// TwinCAT 3 PLC project TwinCAT_OpenFramework_Tests
// Title: TwinCAT Open Framework Tests
// Company: Oleksandr Tiutyk FOP
// Author: Oleksandr Tiutyk
// ProjectVersion: 1.0.13.0
// Description: TwinCAT.OpenFramework regression tests and independent testing framework contract checks
// ProgramVersion: 3.1.4026.28
// libraries:
//   Tc2_Utilities, * (Beckhoff Automation GmbH)
//   [TwinCAT Open Framework JSON], * (Oleksandr Tiutyk FOP)
//   Tc3_JsonXml, * (Beckhoff Automation GmbH)
//   [TwinCAT Open Framework Testing], * (Oleksandr Tiutyk FOP)
//   Tc2_Standard, * (Beckhoff Automation GmbH)
//   Tc2_System, * (Beckhoff Automation GmbH)
//   [TwinCAT Open Framework Devices IO], * (Oleksandr Tiutyk FOP)
//   [TwinCAT Open Framework IO Models], * (Oleksandr Tiutyk FOP)
//   [TwinCAT Open Framework Automation], * (Oleksandr Tiutyk FOP)
//   [TwinCAT Open Framework Collections], * (Oleksandr Tiutyk FOP)
//   [TwinCAT Open Framework Comparison], * (Oleksandr Tiutyk FOP)
//   [TwinCAT Open Framework Core], * (Oleksandr Tiutyk FOP)
//   [TwinCAT Open Framework File System], * (Oleksandr Tiutyk FOP)
//   [TwinCAT Open Framework Loggers], * (Oleksandr Tiutyk FOP)
//   [TwinCAT Open Framework Timers], * (Oleksandr Tiutyk FOP)
//   [TwinCAT Open Framework Tasks], * (Oleksandr Tiutyk FOP)
//   [TwinCAT Open Framework Workflow], * (Oleksandr Tiutyk FOP)
// project tree:
//   Tests/Workflow/ WorkflowBindingTask.TcPOU, ComprehensiveTestWorkflow.TcPOU, RecoveryCatchTestActivity.TcPOU, ThrowingTestActivity.TcPOU, WORKFLOW_COMPREHENSIVE_TEST_SCENARIO.TcDUT, WorkflowComprehensiveTestGroup.TcPOU, WorkflowComprehensiveTestCase.TcPOU, WorkflowComprehensiveTestFixture.TcPOU, WorkflowContractActivity.TcPOU, WorkflowContractWorkflow.TcPOU, WorkflowContractTask.TcPOU, DELAY_PAUSE_TEST_PHASE.TcDUT, WORKFLOW_CONTRACT_TEST_SCENARIO.TcDUT, WorkflowContractTestGroup.TcPOU, WorkflowContractTestCase.TcPOU, WorkflowDelayPauseRemainingTest.TcPOU, WorkflowContractTestFixture.TcPOU
//   / CurrentNamespace.TcGVL, LogFilter.TcPOU, TestAutomationController.TcPOU, MAIN.TcPOU, TestTask.TcTTO, RunnerTestTask.TcTTO
//   Tests/JSON/ JSON_TEST_VALUE.TcDUT, JSON_TEST_SINGLE_VALUE.TcDUT, JSON_TEST_LARGE_VALUE.TcDUT, JsonExtenderProbe.TcPOU, AutomaticJsonRoundTripsAnyStructureTest.TcPOU, AutomaticJsonThrowingAnyRoundTripTest.TcPOU, AutomaticJsonSingleFieldVarInfoRoundTripTest.TcPOU, AutomaticJsonRejectsInvalidArgumentsTest.TcPOU, AutomaticJsonThrowingArgumentCategoriesTest.TcPOU, AutomaticJsonMalformedJsonAndReuseTest.TcPOU, AutomaticJsonWrappedCallbacksTest.TcPOU, AutomaticJsonCallbackContainmentAndReuseTest.TcPOU, AutomaticJsonThrowingCallbackPropagationTest.TcPOU, AutomaticJsonCapacityOverflowAndReuseTest.TcPOU, AutomaticJsonLongUtf8RoundTripTest.TcPOU, AutomaticJsonDecimalPlacesReadbackTest.TcPOU, AutomaticJsonSerializerTestGroup.TcPOU, MockConfigurationWritable.TcPOU, JsonConfigurationWriterTest.TcPOU, JsonConfigurationReaderTest.TcPOU, JsonConfigurationRoundTripTest.TcPOU, JsonConfigurationTestRunner.TcPOU
//   Tests/Collections/Contract/ CollectionCloneProbe.TcPOU, CollectionValidatorProbe.TcPOU, CollectionEqualityProbe.TcPOU, CollectionPredicateProbe.TcPOU, CollectionComparerProbe.TcPOU, COLLECTIONS_CONTRACT_SCENARIO.TcDUT, CollectionsContractTestFixture.TcPOU, CollectionsContractTestCase.TcPOU, CollectionsContractTestGroup.TcPOU, ICollectionSortValue.TcIO, CollectionComparableProbe.TcPOU
//   Tests/Collections/ DictionarySetAndGetTest.TcPOU, DictionaryRemoveTest.TcPOU, DictionaryContainsTest.TcPOU, ByteListTestCase.TcPOU, ByteListLoadFromAnyTest.TcPOU, ByteListIndexedAccessTest.TcPOU, ByteListFindTest.TcPOU, ByteListRemoveValueTest.TcPOU, ByteListRemoveRangeTest.TcPOU, ByteListClearTest.TcPOU, ListAppendTest.TcPOU, ListInsertTest.TcPOU, ListGetAndSetTest.TcPOU, ListFindTest.TcPOU, ListContainsTest.TcPOU, ListContainsGenericTest.TcPOU, ListRemoveFirstTest.TcPOU, ListRemoveMatchedTest.TcPOU, ListRemoveAtTest.TcPOU, ListSwapTest.TcPOU, ListAppendGenericTest.TcPOU, ListInsertGenericTest.TcPOU, ListGetAndSetGenericTest.TcPOU, ListStringPredicate.TcPOU, UniqueDataSetSetAndGetTest.TcPOU, UniqueDataSetRemoveTest.TcPOU, UniqueDataSetContainsTest.TcPOU, StackOwnedObjectCleanupTest.TcPOU, StackValidatorRejectionTest.TcPOU, StackIndexedAccessAndEnumerationTest.TcPOU, StackEmptyAndIndexBoundsTest.TcPOU, StackCopiedAndBorrowedValuesTest.TcPOU, StackContainsTest.TcPOU, StackContainsGenericTest.TcPOU, StackPushAndPeekTest.TcPOU, StackRemoveLastTest.TcPOU
//   Tests/Collections/Dynamic/ DynamicDictionaryClearTest.TcPOU, DynamicDictionaryTestGroup.TcPOU, DynamicByteListTestGroup.TcPOU, DynamicListSortTest.TcPOU, DynamicListClearTest.TcPOU, DynamicListTestGroup.TcPOU, DynamicUniqueDataSetClearTest.TcPOU, DynamicUniqueDataSetTestGroup.TcPOU, DynamicQueueContainsTest.TcPOU, DynamicQueueContainsGenericTest.TcPOU, DynamicQueueEnqueueAndPeekTest.TcPOU, DynamicQueueClearTest.TcPOU, DynamicQueueRemoveFirstTest.TcPOU, DynamicQueueTestGroup.TcPOU, DynamicStackClearTest.TcPOU, DynamicStackGrowthAndInvalidIncrementTest.TcPOU, DynamicStackTestGroup.TcPOU
//   Tests/Collections/Static/ StaticByteListOverflowTest.TcPOU, StaticByteListTestGroup.TcPOU, StaticDictionaryClearTest.TcPOU, StaticDictionaryOverflowTest.TcPOU, StaticDictionaryTestGroup.TcPOU, StaticListSortTest.TcPOU, StaticListClearTest.TcPOU, StaticListOverflowTest.TcPOU, StaticListTestGroup.TcPOU, StaticUniqueDataSetClearTest.TcPOU, StaticUniqueDataSetOverflowTest.TcPOU, StaticUniqueDataSetTestGroup.TcPOU, StaticQueueContainsTest.TcPOU, StaticQueueContainsGenericTest.TcPOU, StaticQueueEnqueueAndPeekTest.TcPOU, StaticQueueClearTest.TcPOU, StaticQueueRemoveFirstTest.TcPOU, StaticQueueOverflowTest.TcPOU, StaticQueueTestGroup.TcPOU, StaticStackClearTest.TcPOU, StaticStackOverflowTest.TcPOU, StaticStackTestGroup.TcPOU
//   Tests/Devices/IO/ RangeAnalogValueConverterTest.TcPOU, RangeAnalogValueConverter16BitTest.TcPOU, RangeAnalogValueConverter32BitTest.TcPOU, RangeAnalogValueConverter32RealTest.TcPOU, AnalogInputConverterProbe.TcPOU, AnalogInputRecoveryProbe.TcPOU, DigitalInputNormallyOpenTest.TcPOU, DigitalInputNormallyClosedTest.TcPOU, DigitalInputUnboundTest.TcPOU, DigitalOutputNormallyOpenTest.TcPOU, DigitalOutputNormallyClosedTest.TcPOU, DirectAnalogValueConverterTest.TcPOU, AnalogInputScalingAndScalarBindingTest.TcPOU, AnalogInputChannelStatusAndErrorReportingTest.TcPOU, AnalogInputConverterRecoveryTest.TcPOU, AnalogInputCriticalConversionErrorTest.TcPOU, AnalogInputStatusWordIsolationTest.TcPOU, AnalogInputStatusBitDecodingTest.TcPOU, AnalogOutputScalingTest.TcPOU, AnalogOutputEqualRawLimitsTest.TcPOU, DynamicRangeAnalogValueConverterTest.TcPOU, StaticConverterCopiesLimitsTest.TcPOU, RangeConverterBoundaryClampingAndZeroDivisionTest.TcPOU, DevicesIOTestGroup.TcPOU, IO_MODELS_TEST_SCENARIO.TcDUT, IIOModelsTestFixture.TcIO, IOModelsTestFixture.TcPOU, IOModelsTestCase.TcPOU, IOModelsTestGroup.TcPOU
//   Tests/Core/ NotImplementedExceptionTest.TcPOU, StandardExceptionChainTest.TcPOU, AggregateExceptionPropagationTest.TcPOU, SavedFrameworkExceptionRethrowTest.TcPOU, SystemExceptionRethrowTest.TcPOU, ExceptionTimestampFormattingTest.TcPOU, SystemExceptionTimestampFormattingTest.TcPOU, SystemExceptionCloneTest.TcPOU, AggregateExceptionCloneTest.TcPOU, ArgumentTypeExceptionCloneTest.TcPOU, ExceptionGraphRejectionTest.TcPOU, AggregateExceptionBoundedMessageTest.TcPOU, ExceptionTestGroup.TcPOU, ObjectExitProbe.TcPOU, GenericLongStringOrderingTest.TcPOU, GenericStringPrefixOrderingTest.TcPOU, GenericNaNOrderingTest.TcPOU, GenericMixedNumericPrecisionTest.TcPOU, GenericConversionPairsTest.TcPOU, SystemTypeClassFormattingTest.TcPOU, SystemTypeClassDiagnosticsTest.TcPOU, GenericBorrowedWritesTest.TcPOU, GenericValueTestGroup.TcPOU, DynamicObjectDisposalTest.TcPOU, ObjectInterfaceAddressTest.TcPOU, StaticObjectReleaseRefusalTest.TcPOU, ObjectLifetimeTestGroup.TcPOU, ExceptionTimestampProbe.TcPOU, RandomRangeTest.TcPOU, RandomAbsoluteDispersionTest.TcPOU, RandomPercentageDispersionTest.TcPOU, RandomTestGroup.TcPOU
//   Tests/Files/ FileManagerStartRefusalProbe.TcPOU, FILE_CALLER_CLEANUP_TEST_PHASE.TcDUT, FILE_OPERATIONS_TEST_PHASE.TcDUT, FILE_BUFFER_TEST_PHASE.TcDUT, FileSystemIntegrationTestGroup.TcPOU, FileByteOperationsTest.TcPOU, FileBinaryBufferMatrixTest.TcPOU, FileCallerExceptionCleanupTest.TcPOU, FileSystemContractTest.TcPOU, FileSystemDefaultNamesTest.TcPOU, FileSystemUnboundContentTest.TcPOU, FileSystemLoadBufferTest.TcPOU, FileSystemQueueBindingTest.TcPOU, FileSystemExceptionCloneTest.TcPOU, FileSystemManagerStartRefusalTest.TcPOU, LexicalPathValidationTest.TcPOU, PATH_VALIDATION_TEST_CASE.TcDUT, FileTestRoot.TcPOU, FILE_TEST_DIRECTORY_PHASE.TcDUT, FileTestDirectory.TcPOU, DIRECTORY_TEST_STEP.TcDUT, DirectoryTest.TcPOU, DirectoryOperationTest.TcPOU, READ_ONLY_FILE_TEST_STEP.TcDUT, FILE_MANAGER_REUSE_TEST_STEP.TcDUT, FILE_TEST_LIFECYCLE.TcDUT, FileContentScenarioTest.TcPOU, FileTextReadWriteTest.TcPOU, FileReadOnlyWriteTest.TcPOU, FileWriteCancellationTest.TcPOU, FileManagerReuseTest.TcPOU, FileContentManagerOperationsTest.TcPOU, OpenMissingFileForReadingTest.TcPOU
//   Tests/Loggers/ LOGGER_DELIVERY_BEHAVIOR.TcDUT, LOGGER_CAPTURED_MESSAGE.TcDUT, LoggerCaptureBackend.TcPOU, LoggerTaskProbe.TcPOU, QueuedLoggerSnapshotTest.TcPOU, LoggerIntegrationTestGroup.TcPOU, EventLoggerCategoryTest.TcPOU, QueuedEventLoggerTest.TcPOU, TextFileLoggerRotationTest.TcPOU, QueuedLoggerCapacityTest.TcPOU, QueuedLoggerDeliveryFailureTest.TcPOU, LoggerFormatterFailureTest.TcPOU, LoggerMetadataAndRecordLimitTest.TcPOU, LoggerTaskDiagnosticsTest.TcPOU, QueuedLoggerAggregateTest.TcPOU, CurrentTaskLoggerRoutingTest.TcPOU, LoggerNonCyclicInitializationTest.TcPOU, LoggerContractTestGroup.TcPOU, LOGGER_DIRECTORY_CLEANUP_PHASE.TcDUT, LoggerTestDirectory.TcPOU, LOGGER_FILE_TEST_PHASE.TcDUT, LoggerRoutingTest.TcPOU
//   Tests/Strings/String/ StringBuilderEmptyTest.TcPOU, StringBuilderContentTest.TcPOU, StringBuilderAssignmentFailureTest.TcPOU, StringBuilderTestGroup.TcPOU, StringFitFormattingTest.TcPOU, StringAppendTest.TcPOU, StringAppendFitTest.TcPOU, StringConcatFitTest.TcPOU, StringContainsTest.TcPOU, StringJoinTest.TcPOU, StringReplacementTest.TcPOU, StringSplitTest.TcPOU, StringTrimTest.TcPOU, StringSeparatorBoundsTest.TcPOU, StringsTestGroup.TcPOU
//   Tests/Strings/WideString/ WideStringBuilderEmptyTest.TcPOU, WideStringBuilderContentTest.TcPOU, WideStringBuilderAssignmentFailureTest.TcPOU, WideStringBuilderTestGroup.TcPOU, WideStringFitFormattingTest.TcPOU, WideStringAppendTest.TcPOU, WideStringAppendFitTest.TcPOU, WideStringConcatFitTest.TcPOU, WideStringContainsTest.TcPOU, WideStringJoinTest.TcPOU, WideStringReplacementTest.TcPOU, WideStringSplitTest.TcPOU, WideStringTrimTest.TcPOU, WideStringSeparatorBoundsTest.TcPOU, WideStringLongFitFormattingTest.TcPOU, WideStringsTestGroup.TcPOU
//   Tests/Tasks/QueueCleanup/ QueueCleanupChild.TcPOU, QueueCleanupQueue.TcPOU, QueueCleanupResource.TcPOU, ThrowingGetMessageException.TcPOU, QUEUE_CLEANUP_TEST_SCENARIO.TcDUT, QUEUE_CLEANUP_TEST_PHASE.TcDUT, TaskQueueCleanupScenarioTest.TcPOU, TaskQueueCleanupTestGroup.TcPOU
//   Tests/Tasks/Sequence/ CounterTask.TcPOU, TaskSequenceFifoTest.TcPOU, TaskQueueEmptyModeTest.TcPOU, TaskSequenceTestGroup.TcPOU
//   Tests/Tasks/Stopping/ TaskStoppingResource.TcPOU, TaskStoppingProbe.TcPOU, TASK_STOPPING_TEST_SCENARIO.TcDUT, TaskStoppingScenarioTest.TcPOU, TaskStoppingTestGroup.TcPOU, TaskStoppingNameTest.TcPOU, TimerRestartProbe.TcPOU, PrepareTimerTestForReuse.TcPOU, TimerMetadataTest.TcPOU, TimerCancelBeforeExecuteTest.TcPOU, TimerResetAfterCompletionTest.TcPOU, TimerPendingRestartTest.TcPOU, TimerRestartResetFailureTest.TcPOU, TimerRestartStartFailureTest.TcPOU, TimerCompletionCallbackTest.TcPOU, TimerCompletionPulseTest.TcPOU, DELAYED_TIMER_TEST_SCENARIO.TcDUT, DelayedTimerObservationTest.TcPOU, TimerIntervalObservationTest.TcPOU, TimerTimingTestGroup.TcPOU, TimerRestartWhileRunningTest.TcPOU
//   Tests/Testing/ AssertionCallerTestRunner.TcPOU, AssertionTestRunner.TcPOU, DeadlineTestRunner.TcPOU, DiagnosticTestRunner.TcPOU, EmptyTestRunner.TcPOU, ExternalRecoveryTestRunner.TcPOU, IsolationTestRunner.TcPOU, MissingChildrenTestRunner.TcPOU, MixedTestRunner.TcPOU, ReporterAbortTestRunner.TcPOU, RootTopologyTestRunner.TcPOU, AssertionIsolationProbe.TcPOU, TestingProbe.TcPOU, ThrowingTestReporter.TcPOU, CapturingAdsLogReporter.TcPOU, ExternalElementProbe.TcPOU, DiagnosticProbe.TcPOU, ASSERTION_PROBE_SCENARIO.TcDUT, AssertionContractProbe.TcPOU, EmptyTestGroup.TcPOU, SingleChildTestGroup.TcPOU, PairTestGroup.TcPOU, FailureTestGroup.TcPOU, NestedFailureTestGroup.TcPOU, DeadlineTestGroup.TcPOU, MissingChildrenTestGroup.TcPOU, TEST_RUNNER_CONTRACT_SCENARIO.TcDUT, TestRunnerContractTest.TcPOU
//   Tests/Tasks/ UnboundTaskStateTest.TcPOU, BoundTaskStateTest.TcPOU, UnboundTaskRunningSubstateTest.TcPOU, BoundTaskRunningSubstateTest.TcPOU, UnboundTaskStopReasonTest.TcPOU, BoundTaskStopReasonTest.TcPOU, TaskReinitViewsTest.TcPOU, TaskNamePreservedByResetTest.TcPOU, TaskLifecycleViewsTestGroup.TcPOU
//   Tests/Automation/ AUTOMATION_COMPONENT_TEST_SCENARIO.TcDUT, AutomationComponentTestGroup.TcPOU, AutomationComponentTestCase.TcPOU, AutomationChildInitializationTimeoutTest.TcPOU, AutomationRunnerObservationTest.TcPOU, AutomationComponentTestFixture.TcPOU, RUNNER_TEST_PHASE.TcDUT, AutomationRunnerTestProgram.TcPOU, AutomationRunnerTestGlobals.TcGVL, MockPluginAutomationController.TcPOU, MockHmiControllerPlugin.TcPOU, MockAutomationController.TcPOU, MockAutomationEvent.TcPOU, MockCompositeAutomationComponent.TcPOU, MockLeafAutomationComponent.TcPOU
//   Version/ Global_Version.TcGVL
// (motion and I/O tree: see PLC project twincat_openframework_core)
// real-time tasks:
//   TASK PlcTask: cycle T#10ms, priority 20, ADS port 350
//   TASK TestTask: cycle T#10ms, priority 1, ADS port 351
//   TASK RunnerTestTask: cycle T#10ms, priority 2, ADS port 354
//   TASK HowToTask: cycle T#10ms, priority 22, ADS port 353
// variable links:

CONFIGURATION TwinCAT_OpenFramework_Tests
    RESOURCE PLC ON TwinCAT3
        TASK TestTask(INTERVAL := T#10ms, PRIORITY := 1);
        TASK RunnerTestTask(INTERVAL := T#10ms, PRIORITY := 2);
        PROGRAM MAIN WITH TestTask : MAIN;
        PROGRAM AutomationRunnerTestProgram WITH RunnerTestTask : AutomationRunnerTestProgram;
    END_RESOURCE
END_CONFIGURATION

// ---- Tests/JSON/JSON_TEST_VALUE.TcDUT
(*
SPDX-FileCopyrightText: © 2026 Oleksandr Tiutyk <trofimich@gmail.com>
SPDX-License-Identifier: MIT
License: https://opensource.org/license/mit
*)

(*!
<summary>Holds a multi-field live value for native JSON round-trip tests.</summary>
*)
TYPE JSON_TEST_VALUE :
STRUCT
	//! <summary>Integer payload with an independent expected value.</summary>
	Number : DINT;
	//! <summary>Boolean payload used to detect incomplete restoration.</summary>
	Ready : BOOL;
END_STRUCT
END_TYPE

// ---- Tests/JSON/JSON_TEST_SINGLE_VALUE.TcDUT
(*
SPDX-FileCopyrightText: © 2026 Oleksandr Tiutyk <trofimich@gmail.com>
SPDX-License-Identifier: MIT
License: https://opensource.org/license/mit
*)

(*!
<summary>Holds a single-field structure for explicit VAR_INFO type resolution.</summary>
*)
TYPE JSON_TEST_SINGLE_VALUE :
STRUCT
	//! <summary>Value restored through the explicit structure type.</summary>
	Number : DINT;
END_STRUCT
END_TYPE

// ---- Tests/JSON/JSON_TEST_LARGE_VALUE.TcDUT
(*
SPDX-FileCopyrightText: © 2026 Oleksandr Tiutyk <trofimich@gmail.com>
SPDX-License-Identifier: MIT
License: https://opensource.org/license/mit
*)

(*!
<summary>Holds long text and a distinct marker for native capacity and encoding tests.</summary>
*)
TYPE JSON_TEST_LARGE_VALUE :
STRUCT
	//! <summary>Uses the framework JSON text capacity in bytes, excluding the terminator.</summary>
	Text : STRING(TOF_Core.Parameters.JSON_DOCUMENT_CHAR_SIZE);
	//! <summary>Independent field that distinguishes the structure from its first member.</summary>
	Marker : DINT;
END_STRUCT
END_TYPE

// ---- Tests/Collections/Contract/COLLECTIONS_CONTRACT_SCENARIO.TcDUT
(*!
<summary>Selects one scenario in the collection contract group.</summary>
<description>
Each value maps to a separately reported single-cycle case.
</description>
*)
{attribute 'qualified_only'}
{attribute 'strict'}
TYPE COLLECTIONS_CONTRACT_SCENARIO :
(
	COPY_FAILURE_PRESERVES_EXCEPTION,
	SECOND_COPY_FAILURE_CLEANUP,
	STATIC_FULL_COPY_CLEANUP,
	BYTE_OVERLAP_AND_BOUNDS,
	BYTE_SIZE_REJECTIONS,
	LIST_OWNERSHIP_REPLACEMENT,
	LIST_REMOVAL_LIMITS,
	SORT_FAILURE_PRESERVES_ENTRIES,
	QUEUE_VALIDATION_AND_GROWTH,
	HASH_COLLISION_GROWTH,
	HASH_EQUALITY_REPRESENTATIONS,
	HASH_OWNERSHIP_ALIASES,
	FULL_STATIC_DUPLICATE_UPDATES,
	QUERY_FAILURE_CLEANUP,
	CONTAINS_COLLECTION_CALLBACK_FAILURES,
	GENERIC_QUERY_RELEASE_MATRIX,
	ALL_CURSOR_CONTRACTS,
	FIXTURE_CLEANUP_AFTER_EXCEPTION,
	DEFAULT_SORT_NUMERIC_BRANCHES,
	DEFAULT_SORT_TEXT_AND_OBJECTS,
	DEFAULT_SORT_EXPLICIT_AND_REJECTION,
	MISSING_CURSOR_SOURCES
);
END_TYPE

// ---- Tests/Devices/IO/IO_MODELS_TEST_SCENARIO.TcDUT
(*!
<summary>Selects one independently reported IO model test scenario.</summary>
*)
{attribute 'qualified_only'}
{attribute 'strict'}
TYPE IO_MODELS_TEST_SCENARIO :
(
	PULSE_TRAIN,
	ENCODER_CHANNELS,
	POWER_MEASUREMENT,
	AUXILIARY,
	COUNTER_AND_LOAD,
	SERIAL_AND_DIAGNOSTICS,
	DISCRETE_CATALOG,
	ANALOG_REPRESENTATIONS,
	DINT_BINDING,
	REAL_BINDING
);
END_TYPE

// ---- Tests/Files/FILE_CALLER_CLEANUP_TEST_PHASE.TcDUT
(*
SPDX-FileCopyrightText: © 2026 Oleksandr Tiutyk <trofimich@gmail.com>
SPDX-License-Identifier: MIT
License: https://opensource.org/license/mit
*)

(*!
<summary>Names the phases of a caught caller-exception cleanup regression.</summary>
*)
{attribute 'qualified_only'}
{attribute 'strict'}
TYPE FILE_CALLER_CLEANUP_TEST_PHASE :
(
	//! <summary>Prepare an exclusively owned scenario directory.</summary>
	PREPARE_DIRECTORY,
	//! <summary>Open a file and leave the manager waiting for future children.</summary>
	OPEN_FILE,
	//! <summary>Observe acquisition and raise a caller-side exception.</summary>
	INJECT_CALLER_EXCEPTION,
	//! <summary>Continue cancellation and stopping after the exception was caught.</summary>
	DRAIN_MANAGER,
	//! <summary>Remove owned artifacts only after release completed.</summary>
	CLEANUP
);
END_TYPE

// ---- Tests/Files/FILE_OPERATIONS_TEST_PHASE.TcDUT
(*
SPDX-FileCopyrightText: © 2026 Oleksandr Tiutyk <trofimich@gmail.com>
SPDX-License-Identifier: MIT
License: https://opensource.org/license/mit
*)

(*!
<summary>Names the phases of a filesystem integration regression.</summary>
*)
{attribute 'qualified_only'}
{attribute 'strict'}
TYPE FILE_OPERATIONS_TEST_PHASE :
(
	//! <summary>prepare directory.</summary>
	PREPARE_DIRECTORY,
	//! <summary>start write.</summary>
	START_WRITE,
	//! <summary>wait for write.</summary>
	WAIT_FOR_WRITE,
	//! <summary>check collisions.</summary>
	CHECK_COLLISIONS,
	//! <summary>wait for collisions.</summary>
	WAIT_FOR_COLLISIONS,
	//! <summary>start load.</summary>
	START_LOAD,
	//! <summary>wait for load.</summary>
	WAIT_FOR_LOAD,
	//! <summary>start rename.</summary>
	START_RENAME,
	//! <summary>wait for rename.</summary>
	WAIT_FOR_RENAME,
	//! <summary>load renamed file.</summary>
	LOAD_RENAMED_FILE,
	//! <summary>wait for renamed load.</summary>
	WAIT_FOR_RENAMED_LOAD,
	//! <summary>start delete.</summary>
	START_DELETE,
	//! <summary>wait for delete.</summary>
	WAIT_FOR_DELETE,
	//! <summary>load deleted file.</summary>
	LOAD_DELETED_FILE,
	//! <summary>wait for missing load.</summary>
	WAIT_FOR_MISSING_LOAD,
	//! <summary>cleanup.</summary>
	CLEANUP
);
END_TYPE

// ---- Tests/Files/FILE_BUFFER_TEST_PHASE.TcDUT
(*
SPDX-FileCopyrightText: © 2026 Oleksandr Tiutyk <trofimich@gmail.com>
SPDX-License-Identifier: MIT
License: https://opensource.org/license/mit
*)

(*!
<summary>Names the phases of a filesystem integration regression.</summary>
*)
{attribute 'qualified_only'}
{attribute 'strict'}
TYPE FILE_BUFFER_TEST_PHASE :
(
	//! <summary>prepare directory.</summary>
	PREPARE_DIRECTORY,
	//! <summary>create file.</summary>
	CREATE_FILE,
	//! <summary>wait for file.</summary>
	WAIT_FOR_FILE,
	//! <summary>start invalid operation.</summary>
	START_INVALID_OPERATION,
	//! <summary>wait for invalid operation.</summary>
	WAIT_FOR_INVALID_OPERATION,
	//! <summary>cleanup.</summary>
	CLEANUP
);
END_TYPE

// ---- Tests/Files/PATH_VALIDATION_TEST_CASE.TcDUT
(*
SPDX-FileCopyrightText: © 2026 Oleksandr Tiutyk <trofimich@gmail.com>
SPDX-License-Identifier: MIT
License: https://opensource.org/license/mit
*)

(*!
<summary>Pairs a path with its expected lexical outcomes for directory and file validation.</summary>
*)
TYPE PATH_VALIDATION_TEST_CASE :
STRUCT
	//! <summary>Null-terminated path passed to each lexical validator.</summary>
	Path : Tc2_System.T_MaxString;
	//! <summary>Expected result from IsValidDirectoryPath.</summary>
	DirectoryAccepted : BOOL;
	//! <summary>Expected result from IsValidFilePath.</summary>
	FileAccepted : BOOL;
END_STRUCT
END_TYPE

// ---- Tests/Files/FILE_TEST_DIRECTORY_PHASE.TcDUT
(*
SPDX-FileCopyrightText: © 2026 Oleksandr Tiutyk <trofimich@gmail.com>
SPDX-License-Identifier: MIT
License: https://opensource.org/license/mit
*)

(*!
<summary>Names preparation and cleanup phases of one exclusively owned file-test directory.</summary>
*)
{attribute 'qualified_only'}
{attribute 'strict'}
TYPE FILE_TEST_DIRECTORY_PHASE :
(
	//! <summary>Create a new directory; an existing entry is a preparation failure.</summary>
	CREATE_DIRECTORY,
	//! <summary>Wait for ordinary creation before establishing ownership.</summary>
	WAIT_FOR_DIRECTORY,
	//! <summary>The scenario exclusively owns its prepared directory.</summary>
	READY,
	//! <summary>Cancel and drain interrupted preparation without guessing ownership.</summary>
	DRAIN_CREATION,
	//! <summary>Attempt deletion of the first registered scenario artifact.</summary>
	DELETE_FIRST_FILE,
	//! <summary>Attempt deletion of the second registered scenario artifact.</summary>
	DELETE_SECOND_FILE,
	//! <summary>Remove the owned directory nonrecursively after file cleanup attempts.</summary>
	REMOVE_DIRECTORY,
	//! <summary>Preparation failed or cleanup attempts finished; inspect result properties.</summary>
	COMPLETE
);
END_TYPE

// ---- Tests/Files/DIRECTORY_TEST_STEP.TcDUT
(*
SPDX-FileCopyrightText: © 2026 Oleksandr Tiutyk <trofimich@gmail.com>
SPDX-License-Identifier: MIT
License: https://opensource.org/license/mit
*)

(*!
<summary>Names the operations and successful completion of DirectoryTest scenarios.</summary>
<description>
Each scenario follows its explicit subset of steps. Advancing requires the expected stop reason and any
existence checks for that step. COMPLETED ends scenario work. Cleanup advances on later test cycles.
The enum is internal to the tests.
</description>
*)
{attribute 'qualified_only'}
{attribute 'strict'}
{attribute 'to_string'}
TYPE DIRECTORY_TEST_STEP :
(
	//! <summary>Create the test directory; success establishes ownership, an existing path causes failure.</summary>
	CREATE_DIRECTORY := 0,
	//! <summary>Verify the newly created test directory exists.</summary>
	CHECK_DIRECTORY_PRESENT,
	//! <summary>Create a child directory inside the owned test directory.</summary>
	CREATE_CHILD_DIRECTORY,
	//! <summary>Verify the first conditional creation produced a child directory.</summary>
	CHECK_CHILD_DIRECTORY_PRESENT,
	//! <summary>Repeat conditional creation while the child directory exists.</summary>
	CREATE_CHILD_DIRECTORY_AGAIN,
	//! <summary>Verify the child directory still exists after repeated creation.</summary>
	CHECK_CHILD_DIRECTORY_PRESENT_AGAIN,
	//! <summary>Require native removal of the nonempty parent directory to fail.</summary>
	REJECT_NONEMPTY_DIRECTORY_REMOVAL,
	//! <summary>Confirm the child still exists after the failed parent removal.</summary>
	CHECK_CHILD_DIRECTORY_RETAINED,
	//! <summary>Remove the owned child directory using conditional removal.</summary>
	REMOVE_CHILD_DIRECTORY,
	//! <summary>Verify that the child directory is absent.</summary>
	CHECK_CHILD_DIRECTORY_ABSENT,
	//! <summary>Repeat conditional removal while the child directory is absent.</summary>
	REMOVE_CHILD_DIRECTORY_AGAIN,
	//! <summary>Verify the child directory is still absent after repeated removal.</summary>
	CHECK_CHILD_DIRECTORY_ABSENT_AGAIN,
	//! <summary>Remove the empty test directory created by this scenario.</summary>
	REMOVE_DIRECTORY,
	//! <summary>Verify the test directory is absent after removal.</summary>
	CHECK_DIRECTORY_ABSENT,
	//! <summary>All scenario operations and postconditions completed successfully.</summary>
	COMPLETED
);
END_TYPE

// ---- Tests/Files/READ_ONLY_FILE_TEST_STEP.TcDUT
(*
SPDX-FileCopyrightText: © 2026 Oleksandr Tiutyk <trofimich@gmail.com>
SPDX-License-Identifier: MIT
License: https://opensource.org/license/mit
*)

(*!
<summary>Names preparation and write-failure checks for a file opened for reading.</summary>
<description>
Steps belong to one test scenario; values are not a serialized protocol. The first member is the initial
preparation step. Test completion and failure cleanup are tracked separately.
</description>
*)
{attribute 'qualified_only'}
{attribute 'strict'}
{attribute 'to_string'}
TYPE READ_ONLY_FILE_TEST_STEP :
(
	CREATE_FILE,
	OPEN_FILE_FOR_READING,
	CHECK_WRITE_FAILURE
);
END_TYPE

// ---- Tests/Files/FILE_MANAGER_REUSE_TEST_STEP.TcDUT
(*
SPDX-FileCopyrightText: © 2026 Oleksandr Tiutyk <trofimich@gmail.com>
SPDX-License-Identifier: MIT
License: https://opensource.org/license/mit
*)

(*!
<summary>Names the two runs and intervening cancellation in the file-manager reuse test.</summary>
<description>
Steps belong to one test scenario; values are not a serialized protocol. The first member is the initial
preparation step. Test completion and failure cleanup are tracked separately.
</description>
*)
{attribute 'qualified_only'}
{attribute 'strict'}
{attribute 'to_string'}
TYPE FILE_MANAGER_REUSE_TEST_STEP :
(
	START_FIRST_WRITE,
	CANCEL_AFTER_WRITE,
	RESET_AND_START_SECOND_FILE,
	CHECK_SECOND_FILE
);
END_TYPE

// ---- Tests/Files/FILE_TEST_LIFECYCLE.TcDUT
(*
SPDX-FileCopyrightText: © 2026 Oleksandr Tiutyk <trofimich@gmail.com>
SPDX-License-Identifier: MIT
License: https://opensource.org/license/mit
*)

(*!
<summary>Separates filesystem scenario execution from cleanup and result reporting.</summary>
<description>
A case remains active while cleanup is pending. Completed drain and cleanup attempts permit FINISHED
and result reporting. Errors remain test failures and do not authorize deleting unowned paths.
Cleanup has no forced deadline. These phases do not guarantee physical close after a native release failure.
</description>
*)
{attribute 'qualified_only'}
{attribute 'strict'}
TYPE FILE_TEST_LIFECYCLE :
(
	//! <summary>Advance the scenario and its deadline until its normal or failed outcome is known.</summary>
	RUNNING_SCENARIO,
	//! <summary>Keep the case active while retained resources stop and owned cleanup attempts finish.</summary>
	CLEANING_UP,
	//! <summary>Cleanup observations were reported for this run.</summary>
	FINISHED
);
END_TYPE

// ---- Tests/Loggers/LOGGER_DELIVERY_BEHAVIOR.TcDUT
(*
SPDX-FileCopyrightText: © 2026 Oleksandr Tiutyk <trofimich@gmail.com>
SPDX-License-Identifier: MIT
License: https://opensource.org/license/mit
*)
(*!
<summary>Selects the deliberate backend outcome used by logger containment tests.</summary>
*)
{attribute 'qualified_only'}
{attribute 'strict'}
TYPE LOGGER_DELIVERY_BEHAVIOR :
(
	ACCEPT,
	REFUSE,
	THROW_EXCEPTION
);
END_TYPE

// ---- Tests/Loggers/LOGGER_CAPTURED_MESSAGE.TcDUT
(*
SPDX-FileCopyrightText: © 2026 Oleksandr Tiutyk <trofimich@gmail.com>
SPDX-License-Identifier: MIT
License: https://opensource.org/license/mit
*)
(*!
<summary>Owns one captured logger call independently of caller buffers.</summary>
*)
TYPE LOGGER_CAPTURED_MESSAGE :
STRUCT
	Category : TOF_Core.LOG_CATEGORY;
	Message : TOF_Core.ERROR_MESSAGE;
	HasMessageNumber : BOOL;
	MessageNumber : ULINT;
END_STRUCT
END_TYPE

// ---- Tests/Loggers/LOGGER_DIRECTORY_CLEANUP_PHASE.TcDUT
(*
SPDX-FileCopyrightText: © 2026 Oleksandr Tiutyk <trofimich@gmail.com>
SPDX-License-Identifier: MIT
License: https://opensource.org/license/mit
*)
(*!
<summary>Identifies owned log discovery, byte readback, deletion and final directory cleanup.</summary>
*)
{attribute 'qualified_only'}
{attribute 'strict'}
TYPE LOGGER_DIRECTORY_CLEANUP_PHASE :
(
	ENUMERATE_FIRST,
	ENUMERATE_WAIT,
	ENUMERATE_NEXT,
	LOAD_FILE,
	WAIT_FOR_LOAD,
	DELETE_FILE,
	WAIT_FOR_DELETE,
	REMOVE_DIRECTORY,
	COMPLETE
);
END_TYPE

// ---- Tests/Loggers/LOGGER_FILE_TEST_PHASE.TcDUT
(*
SPDX-FileCopyrightText: © 2026 Oleksandr Tiutyk <trofimich@gmail.com>
SPDX-License-Identifier: MIT
License: https://opensource.org/license/mit
*)
(*!
<summary>Identifies owned directory preparation, logging, idle observation, stopping and readback phases.</summary>
*)
{attribute 'qualified_only'}
{attribute 'strict'}
TYPE LOGGER_FILE_TEST_PHASE :
(
	PREPARE_DIRECTORY,
	SEND_MESSAGES,
	OBSERVE_IDLE,
	WAIT_FOR_STOP,
	READBACK,
	COMPLETE
);
END_TYPE

// ---- Tests/Tasks/QueueCleanup/QUEUE_CLEANUP_TEST_SCENARIO.TcDUT
(*
SPDX-FileCopyrightText: © 2026 Oleksandr Tiutyk <trofimich@gmail.com>
SPDX-License-Identifier: MIT
License: https://opensource.org/license/mit
*)

(*!
<summary>Selects the faults and observations for a queue cleanup case.</summary>
*)
{attribute 'qualified_only'}
{attribute 'strict'}
TYPE QUEUE_CLEANUP_TEST_SCENARIO :
(
	//! <summary>Completes cleanup, then reuses the same queue and child without injection.</summary>
	DELAYED_CLEANUP_AND_REUSE,
	//! <summary>Raises two further exceptions on cleanup Execute calls.</summary>
	REPEATED_EXECUTE_FAILURE,
	//! <summary>Refuses cancellation by exception twice before accepting it.</summary>
	CANCEL_REQUEST_FAILURE,
	//! <summary>Raises a secondary exception while formatting the original failure.</summary>
	MESSAGE_FORMATTING_FAILURE,
	//! <summary>Requests owner cancellation after the first processing failure.</summary>
	EXTERNAL_CANCEL_DURING_CLEANUP,
	//! <summary>Holds cooperative child cleanup across eight subsequent queue calls.</summary>
	HELD_CLEANUP,
	//! <summary>Requests owner cancellation and injects a terminal parent release failure.</summary>
	EXTERNAL_CANCEL_WITH_RELEASE_FAILURE
);
END_TYPE

// ---- Tests/Tasks/QueueCleanup/QUEUE_CLEANUP_TEST_PHASE.TcDUT
(*
SPDX-FileCopyrightText: © 2026 Oleksandr Tiutyk <trofimich@gmail.com>
SPDX-License-Identifier: MIT
License: https://opensource.org/license/mit
*)

(*!
<summary>Identifies the current queue cleanup test phase.</summary>
*)
{attribute 'qualified_only'}
{attribute 'strict'}
TYPE QUEUE_CLEANUP_TEST_PHASE :
(
	//! <summary>Drive the original failure and child cleanup.</summary>
	FAILURE_RUN,
	//! <summary>Drive the same queue after Reset without a child failure.</summary>
	REUSE_RUN,
	//! <summary>Advance the stopped queue once to check that release is not retried.</summary>
	OBSERVE_FAILED_RELEASE
);
END_TYPE

// ---- Tests/Tasks/Stopping/TASK_STOPPING_TEST_SCENARIO.TcDUT
(*
SPDX-FileCopyrightText: © 2026 Oleksandr Tiutyk <trofimich@gmail.com>
SPDX-License-Identifier: MIT
License: https://opensource.org/license/mit
*)

(*!
<summary>Selects the injection and expected behavior of a task stopping case.</summary>
*)

{attribute 'qualified_only'}
{attribute 'strict'}
TYPE TASK_STOPPING_TEST_SCENARIO :
(
	//! <summary>Completes work and waits for both stopping and release.</summary>
	WORK_DONE,
	//! <summary>Retains the ERROR result and diagnostic after cleanup.</summary>
	WORK_ERROR,
	//! <summary>Retains the ABORTED result and diagnostic after cleanup.</summary>
	WORK_ABORT,
	//! <summary>Defers stopping after a processing exception.</summary>
	WORK_EXCEPTION,
	//! <summary>Uses a named fallback when the processing exception formatter throws.</summary>
	WORK_FORMATTER_EXCEPTION,
	//! <summary>Retries the interrupted stopping hook and preserves the preceding work exception.</summary>
	FIRST_STOPPING_EXCEPTION,
	//! <summary>Interrupts three stopping calls before allowing progress.</summary>
	REPEATED_STOPPING_EXCEPTIONS,
	//! <summary>Produces a named fallback for empty exception text without a bound resource.</summary>
	EMPTY_WORK_EXCEPTION_MESSAGE,
	//! <summary>Cancels a pending acquisition and releases the late acquired resource.</summary>
	CANCEL_DURING_ACQUIRE,
	//! <summary>Cancels before the first Execute and never acquires.</summary>
	CANCEL_BEFORE_ACQUIRE,
	//! <summary>Releases a resource acquired immediately before an exception.</summary>
	ACQUIRE_EXCEPTION_AFTER_OWNERSHIP,
	//! <summary>Stops without release after acquisition is refused.</summary>
	ACQUIRE_EXCEPTION_BEFORE_OWNERSHIP,
	//! <summary>Preserves successful work as the original result when release fails.</summary>
	RELEASE_EXCEPTION,
	//! <summary>Resets from OnAfterStop without reentering work.</summary>
	RESET_IN_NOTIFICATION,
	//! <summary>Refuses Reset with fallback diagnostics and allows a retry.</summary>
	RESET_FORMATTER_EXCEPTION,
	//! <summary>Refuses Start with fallback diagnostics and allows a retry.</summary>
	START_FORMATTER_EXCEPTION
);
END_TYPE

// ---- Tests/Tasks/Stopping/DELAYED_TIMER_TEST_SCENARIO.TcDUT
(*
SPDX-FileCopyrightText: © 2026 Oleksandr Tiutyk <trofimich@gmail.com>
SPDX-License-Identifier: MIT
License: https://opensource.org/license/mit
*)

(*!
<summary>Selects the setup and outcome for a delayed timer observation.</summary>
*)

{attribute 'qualified_only'}
{attribute 'strict'}
TYPE DELAYED_TIMER_TEST_SCENARIO :
(
	//! <summary>Observe natural completion after delaying the first Execute.</summary>
	AFTER_START,
	//! <summary>Request cancellation after the preset but before any Execute.</summary>
	CANCEL_BEFORE_EXECUTE,
	//! <summary>Observe natural completion after restarting an active timer and delaying Execute.</summary>
	AFTER_ACTIVE_RESTART
);
END_TYPE

// ---- Tests/Testing/ASSERTION_PROBE_SCENARIO.TcDUT
(*
SPDX-FileCopyrightText: © 2026 Oleksandr Tiutyk <trofimich@gmail.com>
SPDX-License-Identifier: MIT
License: https://opensource.org/license/mit
*)

(*!
<summary>Selects an independent assertion contract scenario for the regression fixture.</summary>
<description>Each value selects a complete single-cycle body, not a numeric execution phase.</description>
*)

{attribute 'qualified_only'}
{attribute 'strict'}
TYPE ASSERTION_PROBE_SCENARIO :
(
	FLOAT_TOLERANCE,
	INTEGER_EXACT,
	TYPED_LITERALS,
	MESSAGE_CHAIN,
	NEGATIVE_TOLERANCE,
	NAN_TOLERANCE,
	INFINITE_TOLERANCE,
	MESSAGE_RESET,
	POINTERS_AND_STRINGS,
	FIRST_FAILURE,
	SPECIAL_FLOATS,
	OPPOSITE_LIMITS,
	GENERIC_MESSAGE_CHAIN,
	GENERIC_MESSAGE_RESET,
	CONTEXT_TRANSITIONS,
	TYPED_MESSAGE_AFTER_GENERIC,
	GENERIC_MESSAGE_AFTER_TYPED,
	TYPED_MESSAGE_RESET_AFTER_GENERIC,
	INTEGER_FAILURE,
	BITSTRING_FAILURE,
	POINTER_FAILURE,
	STRING_LONG_FAILURE,
	WIDE_STRING_LONG_FAILURE,
	STRING_CONTAINMENT_FAILURE,
	FLOAT_ORDERING_FAILURE,
	FLOAT_EQUALITY_FAILURE,
	TIME_ORDERING_FAILURE
);
END_TYPE

// ---- Tests/Testing/TEST_RUNNER_CONTRACT_SCENARIO.TcDUT
(*!
<summary>Selects the current stage of the independent runner contract suite.</summary>
*)
{attribute 'qualified_only'}
{attribute 'strict'}
TYPE TEST_RUNNER_CONTRACT_SCENARIO :
(
	STARTING,
	ELEMENT_TREE,
	CASE_ISOLATION,
	EMPTY_RUN,
	REPORTER_ABORT,
	DEADLINE,
	GROUP_TOPOLOGY,
	EXTERNAL_RECOVERY,
	DIAGNOSTICS,
	ADS_REPORTER_SUMMARY,
	ASSERTION_CONTRACTS,
	XML_ENCODING,
	RUNNER_TOPOLOGY,
	EXCEPTION_CLASSES,
	CONTEXT_OBJECTS,
	PATHS,
	INDEXED_CHILDREN,
	FINISHED
);
END_TYPE

// ---- Tests/Automation/AUTOMATION_COMPONENT_TEST_SCENARIO.TcDUT
(*!
<summary>Selects one independently reported scenario in the AutomationComponentTest group.</summary>
*)
{attribute 'qualified_only'}
{attribute 'strict'}
TYPE AUTOMATION_COMPONENT_TEST_SCENARIO :
(
	LIFECYCLE_TRANSITIONS,
	ENABLE_DISABLE,
	CHILD_ERROR_POLICY_IGNORE,
	CHILD_ERROR_POLICY_SET_ERROR_AND_CONTINUE,
	CHILD_ERROR_POLICY_SET_ERROR_AND_STOP,
	EVENT_BUBBLING,
	EVENT_BUBBLING_STOP_PROPAGATION,
	EVENT_BROADCASTING,
	INPUT_OUTPUT_PHASES,
	OUTPUT_PHASE_STOP,
	INPUT_PHASE_STOP,
	OUTPUT_PHASE_CONTINUATION,
	PRIMARY_ERROR_BEFORE_LOGGING,
	RESET_CHILD_POLICIES,
	RESET_FROM_STOPPED_HOOK,
	PARENT_VALIDATION,
	DUPLICATE_CHILD,
	MISMATCHED_CHILD_PARENT,
	INITIALIZATION_FAILURE_RESULT,
	INDEXED_LOOKUP_CONTAINMENT,
	CONTROLLER_PLUGIN_RECOVERY,
	RESET_AND_RECOVER_IGNORE_EXCEPTION_POLICY,
	AFTER_CHILDREN_INITIALIZING_AND_TIMEOUT_PROPAGATION,
	DISABLED_CHILD_STOP_RESET_AND_HMI_COMMAND_CONSUMPTION
);
END_TYPE

// ---- Tests/Automation/RUNNER_TEST_PHASE.TcDUT
(*
SPDX-FileCopyrightText: © 2026 Oleksandr Tiutyk <trofimich@gmail.com>
SPDX-License-Identifier: MIT
License: https://opensource.org/license/mit
*)

(*! <summary>Orders the top-level runner calls and publication of their observations.</summary> *)
{attribute 'qualified_only'}
{attribute 'strict'}
TYPE RUNNER_TEST_PHASE :
(
	CHECK_CONSTRUCTION,
	INITIALIZE_ROOTS,
	EXECUTE_ROOTS,
	CHECK_NULL_ROOT,
	CHECK_EMPTY_ROOTS,
	CHECK_DUPLICATE_ROOT,
	PUBLISH_RESULTS,
	FINISHED
);
END_TYPE

// ---- Tests/Workflow/WORKFLOW_COMPREHENSIVE_TEST_SCENARIO.TcDUT
(*!
<summary>Selects one independently reported scenario in the WorkflowComprehensiveTest group.</summary>
*)
{attribute 'qualified_only'}
{attribute 'strict'}
TYPE WORKFLOW_COMPREHENSIVE_TEST_SCENARIO :
(
	END_TO_END_COMPREHENSIVE_SCENARIO,
	WORKFLOW_RESET,
	WORKFLOW_CANCEL,
	PARALLEL_ACTIVITY_WAIT_ALL,
	PARALLEL_ACTIVITY_WAIT_ANY,
	NOT_CONDITION,
	COMPARE_VARIABLE_CONDITION,
	MIXED_NUMERIC_COMPARISON,
	MIXED_TEXT_COMPARISON,
	STANDARD_COMPARISON_FALLBACK,
	INCOMPATIBLE_COMPARISON_PAIRS,
	DIRECT_WORKFLOW_DYNAMIC_CREATION,
	ACTIVITY_VARIABLE_SCOPING_AND_SHADOWING,
	VARIABLE_REGISTRATION_VALIDATION
);
END_TYPE

// ---- Tests/Workflow/DELAY_PAUSE_TEST_PHASE.TcDUT
(*
SPDX-FileCopyrightText: © 2026 Oleksandr Tiutyk <trofimich@gmail.com>
SPDX-License-Identifier: MIT
License: https://opensource.org/license/mit
*)

(*!
<summary>Tracks the cyclic delay pause and reset regression without numerical state flags.</summary>
*)
{attribute 'qualified_only'}
{attribute 'strict'}
TYPE DELAY_PAUSE_TEST_PHASE :
(
	//! <summary>Prepare and start the first active segment.</summary>
	BEFORE_START,
	//! <summary>Accumulate active time before the first pause.</summary>
	FIRST_RUNNING,
	//! <summary>Wait longer than the configured interval while suspended.</summary>
	FIRST_PAUSE,
	//! <summary>Accumulate a second active segment after resuming.</summary>
	SECOND_RUNNING,
	//! <summary>Wait through a second long suspension.</summary>
	SECOND_PAUSE,
	//! <summary>Observe completion against total active time after two pauses.</summary>
	REMAINING_RUNNING,
	//! <summary>Verify a reset starts the full configured interval again.</summary>
	FRESH_RUNNING,
	//! <summary>The scenario has reported its result and must not execute again.</summary>
	FINISHED
);
END_TYPE

// ---- Tests/Workflow/WORKFLOW_CONTRACT_TEST_SCENARIO.TcDUT
(*!
<summary>Selects one independently reported scenario in the WorkflowContractTest group.</summary>
*)
{attribute 'qualified_only'}
{attribute 'strict'}
TYPE WORKFLOW_CONTRACT_TEST_SCENARIO :
(
	ROOT_ASSOCIATION,
	SEQUENCE_TOPOLOGY,
	TRANSITION_DIAGNOSTICS,
	DEPENDENCY_BINDINGS,
	WRITE_CONFIGURATION,
	LOAD_CONFIGURATION,
	OPERATOR_SERIALIZATION,
	DESERIALIZE_NULL_CONTEXT_REJECTION,
	FACTORY_DECLARATIONS,
	ARRAY_VALIDATION,
	WORKFLOW_ISOLATION,
	CONDITION_TOPOLOGY,
	PARENT_SETTERS,
	INITIALIZATION_RETRY,
	BOUNDARY_DIAGNOSTICS,
	INVOKE_CONFIGURATION,
	TASK_FAILURE_DURING_SUSPEND,
	TASK_COMPLETION_DURING_SUSPEND,
	TASK_ABORT_DURING_SUSPEND,
	TASK_RELEASE_FAILURE_DURING_CANCEL,
	CATCH_CLEANUP_BOUNDARY,
	CONCRETE_METADATA,
	VARIABLE_LOOKUP,
	DECLARED_VARIABLE_RESET,
	DECLARED_VARIABLE_VALIDATION,
	CONDITION_SCOPE_PRECEDENCE,
	DELAY_LIFECYCLE
);
END_TYPE

// ---- CurrentNamespace.TcGVL
(*
SPDX-FileCopyrightText: © 2026 Oleksandr Tiutyk <trofimich@gmail.com>
SPDX-License-Identifier: MIT
License: https://opensource.org/license/mit
*)

{attribute 'qualified_only'}
VAR_GLOBAL
	// SA0006: Read-only project namespace string borrowed by tests across tasks.
	{attribute 'analysis' := '-6'}
	Name : STRING := 'TOF_Tests';
END_VAR

// ---- Tests/Automation/AutomationRunnerTestGlobals.TcGVL
(*
SPDX-FileCopyrightText: © 2026 Oleksandr Tiutyk <trofimich@gmail.com>
SPDX-License-Identifier: MIT
License: https://opensource.org/license/mit
*)

(*!
<summary>Provides shared fixtures with early initialization for automation runner tests.</summary>
<description>
Initialized in early slot 40500 so empty sentinel arrays are available during POU variable construction.
</description>
*)

{attribute 'qualified_only'}
{attribute 'global_init_slot' := '40500'}
VAR_GLOBAL CONSTANT
	EmptyComponents : ARRAY [0..-1] OF TOF_Automation.IAutomationComponent := [];
END_VAR

// ---- Version/Global_Version.TcGVL
{attribute 'TcGenerated'}
{attribute 'no-analysis'}
{attribute 'linkalways'}
// This function has been automatically generated from the project information.
VAR_GLOBAL CONSTANT
	{attribute 'const_non_replaced'}
	stLibVersion_TwinCAT_Open_Framework_Tests : ST_LibVersion := (iMajor := 1, iMinor := 0, iBuild := 13, iRevision := 0, nFlags := 0, sVersion := '1.0.13.0');
END_VAR

// ---- Tests/Collections/Contract/ICollectionSortValue.TcIO
(*
SPDX-FileCopyrightText: © 2026 Oleksandr Tiutyk <trofimich@gmail.com>
SPDX-License-Identifier: MIT
License: https://opensource.org/license/mit
*)

(*!
<summary>Exposes a scalar sort key for the collection natural-order fixture.</summary>
<description>
Borrowed interface used to reject unrelated IComparable implementations before reading a sort key.
</description>
*)

INTERFACE ICollectionSortValue EXTENDS TOF_Core.IComparable

(*!
<summary>Returns a copy of the fixture sort key without changing state.</summary>
*)
METHOD GetSortValue : DINT
END_METHOD

END_INTERFACE

// ---- Tests/Devices/IO/IIOModelsTestFixture.TcIO
(*
SPDX-FileCopyrightText: © 2026 Oleksandr Tiutyk <trofimich@gmail.com>
SPDX-License-Identifier: MIT
License: https://opensource.org/license/mit
*)

(*!
<summary>Exposes the IO model scenarios to a single-cycle test case.</summary>
*)

INTERFACE IIOModelsTestFixture

(*!
<summary>Runs one IO model scenario and reports to the current case.</summary>
<description>Use from the owning test task. The fixture never retains assertions.</description>
<param name="scenario">Scenario assigned to the caller.</param>
<param name="assertions">Valid assertion context borrowed from the active case.</param>
*)
METHOD ExecuteScenario
VAR_INPUT
	scenario : IO_MODELS_TEST_SCENARIO;
	assertions : REFERENCE TO TOF_Testing.Assertions;
END_VAR
END_METHOD

END_INTERFACE

// ---- MAIN.TcPOU
(*
SPDX-FileCopyrightText: © 2026 Oleksandr Tiutyk <trofimich@gmail.com>
SPDX-License-Identifier: MIT
License: https://opensource.org/license/mit
*)

(*!
<summary>Runs the test automation controller and reports its lifecycle diagnostics.</summary>
<description>
Services the test runner on each TestTask cycle and reports operational state changes and initialization failures.
</description>
*)

PROGRAM MAIN
VAR_OUTPUT
	TestAutomationUnit : TestAutomationController("TestController");
END_VAR
VAR	
	_AutomationControllers : ARRAY [0..0] OF TOF_Automation.IAutomationComponent := 
	[
		TestAutomationUnit
	];
	_StateInitialized : BOOL;
	_LastState : TOF_Automation.OPERATIONAL_STATE;
	_StateMessage : STRING(255);
	_ErrorMessage : TOF_Core.ERROR_MESSAGE;
	_ReasonMessage : STRING(255);
END_VAR
VAR_OUTPUT
	//! <summary>Installed test filter with a task-local diagnostic probe.</summary>
	DiagnosticLogFilter : LogFilter;
	Runner : TOF_Automation.AutomationRunner(components := _AutomationControllers);
END_VAR

IF Runner.State = TOF_Automation.AUTOMATION_RUNNER_STATE.INITIALIZING THEN
	TOF_Core.LogManager.Filter := DiagnosticLogFilter;	
END_IF

Runner.Execute();

IF Runner.State = TOF_Automation.AUTOMATION_RUNNER_STATE.INVALID THEN
	Tc2_System.ADSLOGSTR(
		msgCtrlMask := Tc2_System.Global_Variables.ADSLOG_MSGTYPE_ERROR,
		msgFmtStr := 'CRITICAL: AutomationRunner is INVALID: %s',
		strArg := TO_STRING(Runner.InitializationErrorMessage)
	);
END_IF

IF NOT _StateInitialized OR_ELSE TestAutomationUnit.OperationalState <> _LastState THEN
	_StateInitialized := TRUE;
	_LastState := TestAutomationUnit.OperationalState;
	_StateMessage := TO_STRING(TestAutomationUnit.OperationalState);

	Tc2_System.ADSLOGSTR(
		msgCtrlMask := Tc2_System.Global_Variables.ADSLOG_MSGTYPE_WARN,
		msgFmtStr := 'STATUS: TestAutomationUnit state changed to: %s',
		strArg := _StateMessage
	);

	IF TestAutomationUnit.OperationalState = TOF_Automation.OPERATIONAL_STATE.STOPPED
		OR_ELSE TestAutomationUnit.OperationalState = TOF_Automation.OPERATIONAL_STATE.INVALID
	THEN
		_ReasonMessage := TO_STRING(TestAutomationUnit.OperationalStateReason);
		_ErrorMessage := TestAutomationUnit.Error.TopMessage;

		Tc2_System.ADSLOGSTR(
			msgCtrlMask := Tc2_System.Global_Variables.ADSLOG_MSGTYPE_ERROR,
			msgFmtStr := 'CRITICAL: TestAutomationUnit stopped/failed. Reason: %s',
			strArg := _ReasonMessage
		);

		Tc2_System.ADSLOGSTR(
			msgCtrlMask := Tc2_System.Global_Variables.ADSLOG_MSGTYPE_ERROR,
			msgFmtStr := 'CRITICAL: TestAutomationUnit error message: %s',
			strArg := TO_STRING(_ErrorMessage)
		);
	END_IF
END_IF

END_PROGRAM

// ---- TestAutomationController.TcPOU
(*
SPDX-FileCopyrightText: © 2026 Oleksandr Tiutyk <trofimich@gmail.com>
SPDX-License-Identifier: MIT
License: https://opensource.org/license/mit
*)

(*!
<summary>Runs the OpenFramework test tree and the independent runner contract suite.</summary>
<description>Instances must not be copied because their test fixtures contain non-copyable state.</description>
*)

{attribute 'no_assign'}
{attribute 'no_explicit_call' := 'do not call this function block directly'}
FUNCTION_BLOCK TestAutomationController EXTENDS TOF_Automation.AutomationController<0>
VAR_STAT
	//! <summary>Class name shared by all instances of this function block.</summary>
	{attribute 'hide'} 
	_ClassName : STRING := __POUNAME();
END_VAR
VAR
	//! <summary>Checks the framework with a separate driver and direct ADS results.</summary>
	_TestRunnerTest : TestRunnerContractTest;

	//! <summary>Owns the I/O symbols and the fixture borrowed by the test runner.</summary>
	_IOModelsTest : IOModelsTestFixture;
	
	//! <summary>Runs the general OpenFramework.Testing regression suites.</summary>
	_JsonConfigurationRunner : JsonConfigurationTestRunner(ioModelsFixture := _IOModelsTest);
END_VAR

PROPERTY Children : REFERENCE TO ARRAY [0.._ChildCount - 1] OF TOF_Automation.IChildAutomationComponent
GET
Children REF= 0;
END_GET
END_PROPERTY

{attribute 'monitoring' := 'call'}
PROPERTY ClassName : REFERENCE TO STRING
GET
ClassName REF= _ClassName;
END_GET
END_PROPERTY

{attribute 'monitoring' := 'call'}
PROPERTY NamespaceName : REFERENCE TO STRING
GET
NamespaceName REF= CurrentNamespace.Name;
END_GET
END_PROPERTY

(*!
<summary>Advances filesystem test-root preparation, the independent contract suite, and the general test tree.</summary>
<description>
One controller task owns FileTestRoot. Suites observe its readiness instead of issuing competing root-create
requests. The independent suite has its own assertions and result reporting. AutomationRunner cleans task
memory after both test paths. Keep calling the controller so root and scenario cleanup can finish.
</description>
*)
METHOD PROTECTED OnBeforeChildrenWorking
VAR
	exceptionCode : __SYSTEM.ExceptionCode;
	exception : TOF_Core.IException;
	lastExMessage : TOF_Core.ERROR_MESSAGE;
	logMessage : STRING(255);
END_VAR
FileTestRoot.Execute();
_TestRunnerTest.Execute();

__TRY
	_JsonConfigurationRunner.Execute(cleanupTaskMemory := FALSE);
__CATCH(exceptionCode)
	exception := TOF_Core.ExceptionManager.GetLastException(
		exceptionCode := exceptionCode,
		catchPointNamespaceName := NamespaceName,
		catchPointPOUName := __POUNAME(),
		catchPointPosition := __POSITION()
	);
	lastExMessage := exception.GetMessage(
		showSource := TRUE,
		timestampDisplayMode := TOF_Core.TIMESTAMP_DISPLAY_MODE.LOCAL
	);
	logMessage := TO_STRING(lastExMessage);

	Tc2_System.ADSLOGSTR(
		msgCtrlMask := Tc2_System.Global_Variables.ADSLOG_MSGTYPE_ERROR,
		msgFmtStr := 'CRITICAL: _JsonConfigurationRunner threw: %s',
		strArg := logMessage
	);

	TOF_Core.ExceptionManager.ReThrowLastException(
		exceptionCode := exceptionCode,
		catchPointNamespaceName := NamespaceName,
		catchPointPOUName := __POUNAME(),
		catchPointPosition := __POSITION()
	);
__ENDTRY
END_METHOD

{attribute 'monitoring' := 'call'}
PROPERTY SelfSize : ULINT
GET
SelfSize := XSIZEOF(THIS^);
END_GET
END_PROPERTY

{attribute 'monitoring' := 'call'}
PROPERTY StartRequest : BOOL
GET
StartRequest := TRUE;
END_GET
END_PROPERTY

END_FUNCTION_BLOCK

// ---- Tests/Testing/TestRunnerContractTest.TcPOU
(*
SPDX-FileCopyrightText: © 2026 Oleksandr Tiutyk <trofimich@gmail.com>
SPDX-License-Identifier: MIT
License: https://opensource.org/license/mit
*)

(*!
<summary>Verifies the testing library with an independent cyclic driver and direct expectations.</summary>
<description>
Runs sixteen scenarios in order with separate inner runners, including deliberately failed inner tests.
Keeps fixtures and the first diagnostic alive across scans. Publishes results directly to the ADS log.
Call Execute once per scan in the owning test task. AutomationRunner owns task memory cleanup.
This suite runs once per application initialization. Do not copy fixture state.
</description>
*)

{attribute 'no_assign'}
{attribute 'no_explicit_call' := 'do not call this function block directly'}
FUNCTION_BLOCK TestRunnerContractTest
VAR_STAT
	{attribute 'hide'}
	_ClassName : STRING := __POUNAME();
END_VAR
VAR CONSTANT
	//! <summary>Number of scenarios scheduled by the independent driver.</summary>
	_TestCount : DINT := 16;
	//! <summary>Maximum calls allowed for the empty runner to report completion.</summary>
	_EmptyScanLimit : UDINT := 16;
	//! <summary>Maximum calls per deadline phase on the configured 10 ms TestTask.</summary>
	_DeadlineScanLimit : UDINT := 32;
END_VAR
VAR_OUTPUT
	//! <summary>Number of completed scenarios with no outer assertion failures.</summary>
	PassedTests : DINT;
	//! <summary>Number of completed scenarios with an outer assertion failure or an unexpected exception.</summary>
	FailedTests : DINT;
	//! <summary>TRUE after every scenario has an outcome and the summary has been published.</summary>
	IsFinished : BOOL;
END_VAR
VAR
	_Scenario : TEST_RUNNER_CONTRACT_SCENARIO;
	_CaseFailed : BOOL;
	_FailureMessage : STRING(255);
END_VAR
VAR
	_Runner : MixedTestRunner;
	_Reporter : TOF_Testing.JUnitXmlReporter;
	_Configured : BOOL;
	_Calls : UDINT;
	_Repeated : BOOL;

	_FailingRun : IsolationTestRunner;
	_PassingRun : AssertionCallerTestRunner;
	_FailureReport : TOF_Testing.JUnitXmlReporter;
	_PassReport : TOF_Testing.JUnitXmlReporter;
	_IsolationConfigured : BOOL;
	_IsolationSecondRun : BOOL;
	_IsolationCalls : UDINT;

	_EmptyRun : EmptyTestRunner;
	_EmptyReport : TOF_Testing.JUnitXmlReporter;
	_EmptyConfigured : BOOL;
	_EmptyCalls : UDINT;
	_AbortRun : ReporterAbortTestRunner;
	_AbortReport : ThrowingTestReporter;
	_InvalidReport : TOF_Testing.JUnitXmlReporter;
	_AbortConfigured : BOOL;
	_AbortCalls : UDINT;
	_AbortPostCalls : UDINT;

	_DeadlineRun : DeadlineTestRunner;
	_DeadlineReport : TOF_Testing.JUnitXmlReporter;
	_DeadlineConfigured : BOOL;
	_DeadlineBusyFailureRun : BOOL;
	_DeadlineCalls : UDINT;
	_ActiveConfigurationChecked : BOOL;

	_DuplicateGroup : PairTestGroup(name := "Duplicates", parent := 0);
	_ParentGroup : SingleChildTestGroup(name := "Parent", parent := _ChildGroup);
	_ChildGroup : SingleChildTestGroup(name := "Child", parent := _ParentGroup);
	_IndexedGroup : PairTestGroup(name := "Indexed children", parent := 0);

	_AbortRecoveryReport : TOF_Testing.JUnitXmlReporter;
	_AbortRecovered : BOOL;
	_ExternalRun : ExternalRecoveryTestRunner;
	_ExternalReport : TOF_Testing.JUnitXmlReporter;
	_ExternalConfigured : BOOL;
	_ExternalRecovered : BOOL;
	_ExternalCalls : UDINT;

	_DiagnosticRun : DiagnosticTestRunner;
	_DiagnosticReport : TOF_Testing.JUnitXmlReporter;
	_DiagnosticConfigured : BOOL;
	_DiagnosticCalls : UDINT;

	_AssertionRun : AssertionTestRunner;
	_AssertionReport : TOF_Testing.JUnitXmlReporter;
	_AssertionsConfigured : BOOL;
	_AssertionCalls : UDINT;

	_XmlReport : TOF_Testing.JUnitXmlReporter;

	_RootTopologyRunner : RootTopologyTestRunner;
	_RootTopologyReport : TOF_Testing.JUnitXmlReporter;
	_RootTopologyConfigured : BOOL;
	_RootTopologyCalls : UDINT;

	_MissingConfigurationGroup : MissingChildrenTestGroup(name := "Missing configuration", parent := 0);
	_MissingConfigurationRunner : MissingChildrenTestRunner;
	_ExceptionAdsReporter : TOF_Testing.AdsLogReporter;
	_AdsSummaryReporter : CapturingAdsLogReporter;

	//! <summary>Synthetic Parent chains for path observation only; these fixtures are not executed as trees.</summary>
	_PathRoot : EmptyTestGroup(
		name := "AAAAAAAAAAAAAAAAAAAAAAAAAAAAAAAAAAAAAAAAAAAAAAAAAAAAAAAAAAAAAAAAAAAAAAAAAAAAAAAA",
		parent := 0
	);
	_PathSecond : EmptyTestGroup(
		name := "BBBBBBBBBBBBBBBBBBBBBBBBBBBBBBBBBBBBBBBBBBBBBBBBBBBBBBBBBBBBBBBBBBBBBBBBBBBBBBBB",
		parent := _PathRoot
	);
	_PathThird : EmptyTestGroup(
		name := "CCCCCCCCCCCCCCCCCCCCCCCCCCCCCCCCCCCCCCCCCCCCCCCCCCCCCCCCCCCCCCCCCCCCCCCCCCCCCCCC",
		parent := _PathSecond
	);
	_PathFourth : EmptyTestGroup(
		name := "DDDDDDDDDDDDDDDDDDDDDDDDDDDDDDDDDDDDDDDDDDDDDDDDDDDDDDDDDDDDDDDDDDDDDDDDDDDDDDDD",
		parent := _PathThird
	);
	_PathEmpty : EmptyTestGroup(name := "", parent := _PathRoot);
	_PathUnicode : TestingProbe(name := "Ω", parent := _PathEmpty);
	//! <summary>Supplies 81 characters to exercise ordinary truncation at the 80-character name input.</summary>
	_PathLongNameInput : WSTRING(81) := "AAAAAAAAAAAAAAAAAAAAAAAAAAAAAAAAAAAAAAAAAAAAAAAAAAAAAAAAAAAAAAAAAAAAAAAAAAAAAAAAB";
	_PathLongName : EmptyTestGroup(
		name := _PathLongNameInput,
		parent := 0
	);
	_ReportPathRoot : EmptyTestGroup(name := "Report root", parent := 0);
	_ReportPathMiddle : EmptyTestGroup(name := "Middle", parent := _ReportPathRoot);
	_ReportPathInner : EmptyTestGroup(name := "Inner", parent := _ReportPathMiddle);
	_PathReport : TOF_Testing.JUnitXmlReporter;
	_MetadataBoolAssertionContext : TOF_Testing.BoolAssertionContext;
	_MetadataByteAssertionContext : TOF_Testing.ByteAssertionContext;
	_MetadataDateAssertionContext : TOF_Testing.DateAssertionContext;
	_MetadataDateTimeAssertionContext : TOF_Testing.DateTimeAssertionContext;
	_MetadataDIntAssertionContext : TOF_Testing.DIntAssertionContext;
	_MetadataDWordAssertionContext : TOF_Testing.DWordAssertionContext;
	_MetadataIntAssertionContext : TOF_Testing.IntAssertionContext;
	_MetadataLIntAssertionContext : TOF_Testing.LIntAssertionContext;
	_MetadataLongDateAssertionContext : TOF_Testing.LongDateAssertionContext;
	_MetadataLongDateTimeAssertionContext : TOF_Testing.LongDateTimeAssertionContext;
	_MetadataLongRealAssertionContext : TOF_Testing.LongRealAssertionContext;
	_MetadataLongTimeAssertionContext : TOF_Testing.LongTimeAssertionContext;
	_MetadataLongTimeOfDayAssertionContext : TOF_Testing.LongTimeOfDayAssertionContext;
	_MetadataLWordAssertionContext : TOF_Testing.LWordAssertionContext;
	_MetadataPointerAssertionContext : TOF_Testing.PointerAssertionContext;
	_MetadataRealAssertionContext : TOF_Testing.RealAssertionContext;
	_MetadataSIntAssertionContext : TOF_Testing.SIntAssertionContext;
	_MetadataStringAssertionContext : TOF_Testing.StringAssertionContext;
	_MetadataTimeAssertionContext : TOF_Testing.TimeAssertionContext;
	_MetadataTimeOfDayAssertionContext : TOF_Testing.TimeOfDayAssertionContext;
	_MetadataUDIntAssertionContext : TOF_Testing.UDIntAssertionContext;
	_MetadataUIntAssertionContext : TOF_Testing.UIntAssertionContext;
	_MetadataULIntAssertionContext : TOF_Testing.ULIntAssertionContext;
	_MetadataUSIntAssertionContext : TOF_Testing.USIntAssertionContext;
	_MetadataWideStringAssertionContext : TOF_Testing.WideStringAssertionContext;
	_MetadataWordAssertionContext : TOF_Testing.WordAssertionContext;
	_OtherBoolContext : TOF_Testing.BoolAssertionContext;
END_VAR

(*!
<summary>Advances one scenario and reports its outcome after completion.</summary>
<description>
Retains the first failed expectation across pending cycles. An unexpected exception fails the active scenario.
Checks the allocation latch outside the recovery block. The caller owns task memory cleanup.
Returns immediately after all scenarios finish and publishes exactly one summary per initialization.
</description>
*)
METHOD Execute
VAR
	caseName : STRING(80);
	nextScenario : TEST_RUNNER_CONTRACT_SCENARIO;
	completed : BOOL;
	exceptionCode : __SYSTEM.ExceptionCode;
END_VAR
IF IsFinished THEN
	RETURN;
END_IF

IF _Scenario = TEST_RUNNER_CONTRACT_SCENARIO.STARTING THEN
	logResult(isError := FALSE, message := TOF_Core.Strings.Concat255('Starting ', TO_STRING(_TestCount), ' tests'));
	_Scenario := TEST_RUNNER_CONTRACT_SCENARIO.ELEMENT_TREE;

	RETURN;
END_IF

__TRY
	CASE _Scenario OF
		TEST_RUNNER_CONTRACT_SCENARIO.ELEMENT_TREE:
			caseName := 'Element tree, lifecycle, repeated run and JUnit';
			nextScenario := TEST_RUNNER_CONTRACT_SCENARIO.CASE_ISOLATION;
			completed := runAndCheck();

		TEST_RUNNER_CONTRACT_SCENARIO.CASE_ISOLATION:
			caseName := 'Each failure belongs to its receiving case';
			nextScenario := TEST_RUNNER_CONTRACT_SCENARIO.EMPTY_RUN;
			completed := checkCaseIsolation();

		TEST_RUNNER_CONTRACT_SCENARIO.EMPTY_RUN:
			caseName := 'An empty root passes with zero tests';
			nextScenario := TEST_RUNNER_CONTRACT_SCENARIO.REPORTER_ABORT;
			completed := checkEmptyRun();

		TEST_RUNNER_CONTRACT_SCENARIO.REPORTER_ABORT:
			caseName := 'A throwing reporter aborts without retry';
			nextScenario := TEST_RUNNER_CONTRACT_SCENARIO.DEADLINE;
			completed := checkReporterAbort();

		TEST_RUNNER_CONTRACT_SCENARIO.DEADLINE:
			caseName := 'A pending multi-cycle test fails at its deadline';
			nextScenario := TEST_RUNNER_CONTRACT_SCENARIO.GROUP_TOPOLOGY;
			completed := checkDeadline();

		TEST_RUNNER_CONTRACT_SCENARIO.GROUP_TOPOLOGY:
			caseName := 'Static group topology is validated before child callbacks';
			nextScenario := TEST_RUNNER_CONTRACT_SCENARIO.EXTERNAL_RECOVERY;
			completed := checkTopology();

		TEST_RUNNER_CONTRACT_SCENARIO.EXTERNAL_RECOVERY:
			caseName := 'External abort recovery can be retried for the same static tree';
			nextScenario := TEST_RUNNER_CONTRACT_SCENARIO.DIAGNOSTICS;
			completed := checkExternalRecovery();

		TEST_RUNNER_CONTRACT_SCENARIO.DIAGNOSTICS:
			caseName := 'Native and framework diagnostics outlive their exception objects';
			nextScenario := TEST_RUNNER_CONTRACT_SCENARIO.ADS_REPORTER_SUMMARY;
			completed := checkDiagnostics();

		TEST_RUNNER_CONTRACT_SCENARIO.ADS_REPORTER_SUMMARY:
			caseName := 'ADS summary retains first failure and resets on the next run';
			nextScenario := TEST_RUNNER_CONTRACT_SCENARIO.ASSERTION_CONTRACTS;
			completed := checkAdsReporterSummary();

		TEST_RUNNER_CONTRACT_SCENARIO.ASSERTION_CONTRACTS:
			caseName := 'Independent contexts, typed predicates, snapshots and chain diagnostics';
			nextScenario := TEST_RUNNER_CONTRACT_SCENARIO.XML_ENCODING;
			completed := checkAssertionContracts();

		TEST_RUNNER_CONTRACT_SCENARIO.XML_ENCODING:
			caseName := 'JUnit preserves long text and replaces forbidden Unicode sequences';
			nextScenario := TEST_RUNNER_CONTRACT_SCENARIO.RUNNER_TOPOLOGY;
			completed := checkXmlEncoding();

		TEST_RUNNER_CONTRACT_SCENARIO.RUNNER_TOPOLOGY:
			caseName := 'Static runner validates roots at startup and executes without rescanning';
			nextScenario := TEST_RUNNER_CONTRACT_SCENARIO.EXCEPTION_CLASSES;
			completed := checkRunnerTopology();

		TEST_RUNNER_CONTRACT_SCENARIO.EXCEPTION_CLASSES:
			caseName := 'Missing static storage is diagnosed before child access';
			nextScenario := TEST_RUNNER_CONTRACT_SCENARIO.CONTEXT_OBJECTS;
			completed := checkExceptionClasses();

		TEST_RUNNER_CONTRACT_SCENARIO.CONTEXT_OBJECTS:
			caseName := 'Typed contexts and concrete runner expose Object metadata and identity';
			nextScenario := TEST_RUNNER_CONTRACT_SCENARIO.PATHS;
			completed := checkContextObjects();

		TEST_RUNNER_CONTRACT_SCENARIO.PATHS:
			caseName := 'Paths follow live Parent links without Reset context';
			nextScenario := TEST_RUNNER_CONTRACT_SCENARIO.INDEXED_CHILDREN;
			completed := checkPaths();

		TEST_RUNNER_CONTRACT_SCENARIO.INDEXED_CHILDREN:
			caseName := 'Indexed children preserve order and reject missing storage or invalid indices';
			nextScenario := TEST_RUNNER_CONTRACT_SCENARIO.FINISHED;
			completed := checkIndexedChildren();
	ELSE
		caseName := 'Scenario selection';
		nextScenario := TEST_RUNNER_CONTRACT_SCENARIO.FINISHED;
		expect(condition := FALSE, message := 'Invalid scenario selection');
		completed := TRUE;
	END_CASE
__CATCH(exceptionCode)
	expect(
		condition := FALSE,
		message := TOF_Core.Strings.Concat255('Unexpected PLC exception ', TO_STRING(exceptionCode))
	);
	completed := TRUE;
__ENDTRY

TOF_Core.DynamicMemoryManager.RaiseIfAllocationFailed();

IF NOT completed THEN
	RETURN;
END_IF

IF _CaseFailed THEN
	FailedTests := FailedTests + 1;
	logResult(
		isError := TRUE,
		message := TOF_Core.Strings.Concat255(caseName, ': ', _FailureMessage)
	);
ELSE
	PassedTests := PassedTests + 1;
END_IF

_CaseFailed := FALSE;
_FailureMessage := '';
_Scenario := nextScenario;

IF _Scenario = TEST_RUNNER_CONTRACT_SCENARIO.FINISHED THEN
	logResult(
		isError := FailedTests <> 0,
		message := TOF_Core.Strings.Concat255(
			'Finished: ',
			TO_STRING(PassedTests),
			' passed, ',
			TO_STRING(FailedTests),
			' failed'
		)
	);
	IsFinished := TRUE;
END_IF
END_METHOD

(*!
<summary>Copies the first diagnostic when an expectation fails.</summary>
<param name="condition">TRUE when the expectation holds.</param>
<param name="message">Description of the failed expectation.</param>
*)
METHOD PRIVATE expect
VAR_INPUT
	condition : BOOL;
	message : STRING(255);
END_VAR
IF NOT condition AND_THEN NOT _CaseFailed THEN
	_CaseFailed := TRUE;
	_FailureMessage := message;
END_IF
END_METHOD

(*!
<summary>Checks that a predicate is false.</summary>
<param name="condition">Predicate that must be FALSE.</param>
<param name="message">Description of the failed expectation.</param>
*)
METHOD PRIVATE expectFalse
VAR_INPUT
	condition : BOOL;
	message : STRING(255);
END_VAR
expect(condition := NOT condition, message := message);
END_METHOD

(*!
<summary>Compares two DINT values and records differences.</summary>
<param name="expected">Expected value determined by the scenario.</param>
<param name="actual">Observed value.</param>
<param name="message">Description of the failed expectation.</param>
*)
METHOD PRIVATE expectDInt
VAR_INPUT
	expected : DINT;
	actual : DINT;
	message : STRING(255);
END_VAR
IF actual <> expected AND_THEN NOT _CaseFailed THEN
	expect(
		condition := FALSE,
		message := TOF_Core.Strings.Concat255(
			message,
			' (expected ',
			TO_STRING(expected),
			', actual ',
			TO_STRING(actual),
			')'
		)
	);
END_IF
END_METHOD

(*!
<summary>Compares two UDINT values and records differences.</summary>
<param name="expected">Expected value determined by the scenario.</param>
<param name="actual">Observed value.</param>
<param name="message">Description of the failed expectation.</param>
*)
METHOD PRIVATE expectUDInt
VAR_INPUT
	expected : UDINT;
	actual : UDINT;
	message : STRING(255);
END_VAR
IF actual <> expected AND_THEN NOT _CaseFailed THEN
	expect(
		condition := FALSE,
		message := TOF_Core.Strings.Concat255(
			message,
			' (expected ',
			TO_STRING(expected),
			', actual ',
			TO_STRING(actual),
			')'
		)
	);
END_IF
END_METHOD

(*!
<summary>Publishes a diagnostic without using the library under test.</summary>
<param name="isError">TRUE for scenario errors and failed summaries.</param>
<param name="message">Diagnostic to publish.</param>
*)
METHOD PRIVATE logResult
VAR_INPUT
	isError : BOOL;
	message : STRING(255);
END_VAR
VAR
	severity : DWORD;
END_VAR
severity := SEL(
	isError,
	Tc2_System.Global_Variables.ADSLOG_MSGTYPE_HINT,
	Tc2_System.Global_Variables.ADSLOG_MSGTYPE_ERROR
);

Tc2_System.ADSLOGSTR(
	msgCtrlMask := severity OR Tc2_System.Global_Variables.ADSLOG_MSGTYPE_LOG,
	msgFmtStr := '[TestRunnerContractTest] %s',
	strArg := message
);
END_METHOD

(*!
<summary>Checks a caught failure through its dedicated exception interface before task cleanup.</summary>
<description>Only borrows the exception during this call; no exception reference survives the test cycle.</description>
*)
METHOD PRIVATE assertCaughtExceptionType
VAR_INPUT
	exceptionCode : __SYSTEM.ExceptionCode;
	expectedTypeName : STRING;
END_VAR
VAR
	exception : TOF_Core.IException;
	standardException : TOF_Core.IStandardException;
	argumentNotSpecified : TOF_Core.IArgumentNotSpecifiedException;
	memberNotSpecified : TOF_Core.IDataMemberNotSpecifiedException;
	argumentValueNotSupported : TOF_Core.IArgumentValueNotSupportedException;
	argumentOutOfRange : TOF_Core.IArgumentOutOfRangeException;
	matchesType : BOOL;
END_VAR
exception := TOF_Core.ExceptionManager.GetLastException(
	exceptionCode := exceptionCode,
	catchPointNamespaceName := CurrentNamespace.Name,
	catchPointPOUName := __POUNAME(),
	catchPointPosition := __POSITION()
);
expect(condition := exception <> 0, message := 'Caught failure exposes its exception payload');

IF exception = 0 THEN
	RETURN;
END_IF

IF expectedTypeName = 'StandardException' THEN
	matchesType := __QUERYINTERFACE(exception, standardException);
ELSIF expectedTypeName = 'ArgumentNotSpecifiedException' THEN
	matchesType := __QUERYINTERFACE(exception, argumentNotSpecified);
ELSIF expectedTypeName = 'DataMemberNotSpecifiedException' THEN
	matchesType := __QUERYINTERFACE(exception, memberNotSpecified);
ELSIF expectedTypeName = 'ArgumentValueNotSupportedException' THEN
	matchesType := __QUERYINTERFACE(exception, argumentValueNotSupported);
ELSIF expectedTypeName = 'ArgumentOutOfRangeException' THEN
	matchesType := __QUERYINTERFACE(exception, argumentOutOfRange);
END_IF

expect(condition := matchesType, message := 'Exception interface matches the expected failure category');
END_METHOD

(*!
<summary>Checks concrete metadata through a borrowed Object interface.</summary>
<description>Checks namespace, class, size and address separately with distinct failure diagnostics.</description>
<param name="object">Live instance whose metadata is read without preparation.</param>
<param name="expectedNamespaceName">Namespace of the project declaring the concrete type.</param>
<param name="expectedClassName">Concrete context class name.</param>
<param name="expectedSize">Compiler-reported size of the complete concrete context.</param>
<param name="expectedAddress">Address of the concrete context, without ownership transfer.</param>
*)
METHOD PRIVATE assertObjectMetadata
VAR_INPUT
	object : TOF_Core.IObject;
	expectedNamespaceName : STRING;
	expectedClassName : STRING;
	expectedSize : ULINT;
	expectedAddress : PVOID;
END_VAR
expect(condition := object <> 0, message := expectedClassName);

IF object = 0 THEN
	RETURN;
END_IF

expect(
	condition := object.ClassName = expectedClassName,
	message := TOF_Core.Strings.Concat255(expectedClassName, ': ClassName')
);
expect(
	condition := object.NamespaceName = expectedNamespaceName,
	message := TOF_Core.Strings.Concat255(expectedClassName, ': NamespaceName')
);
expect(
	condition := object.SelfSize = expectedSize,
	message := TOF_Core.Strings.Concat255(expectedClassName, ': SelfSize')
);
expect(
	condition := object.SelfAddress = expectedAddress,
	message := TOF_Core.Strings.Concat255(expectedClassName, ': SelfAddress')
);
END_METHOD

(*!
<summary>Checks independent typed and generic contexts, native predicates and chain-wide diagnostics.</summary>
<description>Configures the persistent output probes through a local reference without copying them.
Returns TRUE when all observations for this scenario are complete.
</description>
*)
METHOD PRIVATE checkAssertionContracts : BOOL
VAR
	probe : REFERENCE TO AssertionContractProbe;
END_VAR
IF NOT _AssertionsConfigured THEN
	probe REF= _AssertionRun.Assertion0;
	probe.Scenario := ASSERTION_PROBE_SCENARIO.FLOAT_TOLERANCE;
	probe REF= _AssertionRun.Assertion1;
	probe.Scenario := ASSERTION_PROBE_SCENARIO.INTEGER_EXACT;
	probe REF= _AssertionRun.Assertion2;
	probe.Scenario := ASSERTION_PROBE_SCENARIO.TYPED_LITERALS;
	probe REF= _AssertionRun.Assertion3;
	probe.Scenario := ASSERTION_PROBE_SCENARIO.MESSAGE_CHAIN;
	probe REF= _AssertionRun.Assertion4;
	probe.Scenario := ASSERTION_PROBE_SCENARIO.NEGATIVE_TOLERANCE;
	probe REF= _AssertionRun.Assertion5;
	probe.Scenario := ASSERTION_PROBE_SCENARIO.NAN_TOLERANCE;
	probe REF= _AssertionRun.Assertion6;
	probe.Scenario := ASSERTION_PROBE_SCENARIO.INFINITE_TOLERANCE;
	probe REF= _AssertionRun.Assertion7;
	probe.Scenario := ASSERTION_PROBE_SCENARIO.MESSAGE_RESET;
	probe REF= _AssertionRun.Assertion8;
	probe.Scenario := ASSERTION_PROBE_SCENARIO.POINTERS_AND_STRINGS;
	probe REF= _AssertionRun.Assertion9;
	probe.Scenario := ASSERTION_PROBE_SCENARIO.FIRST_FAILURE;
	probe REF= _AssertionRun.Assertion10;
	probe.Scenario := ASSERTION_PROBE_SCENARIO.SPECIAL_FLOATS;
	probe REF= _AssertionRun.Assertion11;
	probe.Scenario := ASSERTION_PROBE_SCENARIO.OPPOSITE_LIMITS;
	probe REF= _AssertionRun.Assertion12;
	probe.Scenario := ASSERTION_PROBE_SCENARIO.GENERIC_MESSAGE_CHAIN;
	probe REF= _AssertionRun.Assertion13;
	probe.Scenario := ASSERTION_PROBE_SCENARIO.GENERIC_MESSAGE_RESET;
	probe REF= _AssertionRun.Assertion14;
	probe.Scenario := ASSERTION_PROBE_SCENARIO.CONTEXT_TRANSITIONS;
	probe REF= _AssertionRun.Assertion15;
	probe.Scenario := ASSERTION_PROBE_SCENARIO.TYPED_MESSAGE_AFTER_GENERIC;
	probe REF= _AssertionRun.Assertion16;
	probe.Scenario := ASSERTION_PROBE_SCENARIO.GENERIC_MESSAGE_AFTER_TYPED;
	probe REF= _AssertionRun.Assertion17;
	probe.Scenario := ASSERTION_PROBE_SCENARIO.TYPED_MESSAGE_RESET_AFTER_GENERIC;
	probe REF= _AssertionRun.Assertion18;
	probe.Scenario := ASSERTION_PROBE_SCENARIO.INTEGER_FAILURE;
	probe REF= _AssertionRun.Assertion19;
	probe.Scenario := ASSERTION_PROBE_SCENARIO.BITSTRING_FAILURE;
	probe REF= _AssertionRun.Assertion20;
	probe.Scenario := ASSERTION_PROBE_SCENARIO.POINTER_FAILURE;
	probe REF= _AssertionRun.Assertion21;
	probe.Scenario := ASSERTION_PROBE_SCENARIO.STRING_LONG_FAILURE;
	probe REF= _AssertionRun.Assertion22;
	probe.Scenario := ASSERTION_PROBE_SCENARIO.WIDE_STRING_LONG_FAILURE;
	probe REF= _AssertionRun.Assertion23;
	probe.Scenario := ASSERTION_PROBE_SCENARIO.STRING_CONTAINMENT_FAILURE;
	probe REF= _AssertionRun.Assertion24;
	probe.Scenario := ASSERTION_PROBE_SCENARIO.FLOAT_ORDERING_FAILURE;
	probe REF= _AssertionRun.Assertion25;
	probe.Scenario := ASSERTION_PROBE_SCENARIO.FLOAT_EQUALITY_FAILURE;
	probe REF= _AssertionRun.Assertion26;
	probe.Scenario := ASSERTION_PROBE_SCENARIO.TIME_ORDERING_FAILURE;
	_AssertionRun.Reporter := _AssertionReport;
	_AssertionsConfigured := TRUE;
END_IF

_AssertionRun.Execute(cleanupTaskMemory := FALSE);
_AssertionCalls := _AssertionCalls + 1;

IF NOT _AssertionRun.IsFinished AND_THEN _AssertionCalls < 32 THEN
	RETURN;
END_IF

expect(condition := _AssertionRun.IsFinished, message := 'Twenty-seven assertion leaves finish within 32 scans');
expectDInt(expected := 27, actual := _AssertionRun.TotalTests, message := 'Every assertion scenario executes');
expectDInt(
	expected := 7,
	actual := _AssertionRun.PassedTests,
	message := 'Seven supported assertion scenarios pass'
);
expectDInt(
	expected := 20,
	actual := _AssertionRun.FailedTests,
	message := 'Twenty deliberate failures are recorded'
);
expect(
	condition := _AssertionRun.Assertion0.Outcome = TOF_Testing.TEST_OUTCOME.PASSED,
	message := 'Assertion scenario 0 has its expected passed outcome'
);
expect(
	condition := _AssertionRun.Assertion1.Outcome = TOF_Testing.TEST_OUTCOME.PASSED,
	message := 'Assertion scenario 1 has its expected passed outcome'
);
expect(
	condition := _AssertionRun.Assertion2.Outcome = TOF_Testing.TEST_OUTCOME.PASSED,
	message := 'Assertion scenario 2 has its expected passed outcome'
);
expect(
	condition := _AssertionRun.Assertion3.Outcome = TOF_Testing.TEST_OUTCOME.FAILED,
	message := 'Assertion scenario 3 has its expected failed outcome'
);
expect(
	condition := _AssertionRun.Assertion4.Outcome = TOF_Testing.TEST_OUTCOME.FAILED,
	message := 'Assertion scenario 4 has its expected failed outcome'
);
expect(
	condition := _AssertionRun.Assertion5.Outcome = TOF_Testing.TEST_OUTCOME.FAILED,
	message := 'Assertion scenario 5 has its expected failed outcome'
);
expect(
	condition := _AssertionRun.Assertion6.Outcome = TOF_Testing.TEST_OUTCOME.FAILED,
	message := 'Assertion scenario 6 has its expected failed outcome'
);
expect(
	condition := _AssertionRun.Assertion7.Outcome = TOF_Testing.TEST_OUTCOME.FAILED,
	message := 'Assertion scenario 7 has its expected failed outcome'
);
expect(
	condition := _AssertionRun.Assertion8.Outcome = TOF_Testing.TEST_OUTCOME.PASSED,
	message := 'Assertion scenario 8 has its expected passed outcome'
);
expect(
	condition := _AssertionRun.Assertion9.Outcome = TOF_Testing.TEST_OUTCOME.FAILED,
	message := 'Assertion scenario 9 has its expected failed outcome'
);
expect(
	condition := _AssertionRun.Assertion10.Outcome = TOF_Testing.TEST_OUTCOME.PASSED,
	message := 'Assertion scenario 10 has its expected passed outcome'
);
expect(
	condition := _AssertionRun.Assertion11.Outcome = TOF_Testing.TEST_OUTCOME.PASSED,
	message := 'Assertion scenario 11 has its expected passed outcome'
);
expect(
	condition := _AssertionRun.Assertion12.Outcome = TOF_Testing.TEST_OUTCOME.FAILED,
	message := 'Assertion scenario 12 has its expected failed outcome'
);
expect(
	condition := _AssertionRun.Assertion13.Outcome = TOF_Testing.TEST_OUTCOME.FAILED,
	message := 'Assertion scenario 13 has its expected failed outcome'
);
expect(
	condition := _AssertionRun.Assertion9.FailureMessage = "First diagnostic",
	message := 'Later assertion and teardown exception preserve the first failure'
);
expect(
	condition := TOF_Core.WideStrings.Contains(
		stringToSearchIn := _AssertionRun.Assertion3.FailureMessage,
		stringToFind := "Chain diagnostic: Expected value < "
	),
	message := 'The message survives a successful assertion in the same typed chain'
);
expect(
	condition := NOT TOF_Core.WideStrings.Contains(
		stringToSearchIn := _AssertionRun.Assertion7.FailureMessage,
		stringToFind := "Previous diagnostic"
	),
	message := 'Omitting the typed entry message clears the previous prefix'
);
expect(
	condition := TOF_Core.WideStrings.Contains(
		stringToSearchIn := _AssertionRun.Assertion12.FailureMessage,
		stringToFind := "Generic chain diagnostic: Expected value < "
	),
	message := 'Borrowed assertions retain the same chain-wide message contract'
);
expect(
	condition := NOT TOF_Core.WideStrings.Contains(
		stringToSearchIn := _AssertionRun.Assertion13.FailureMessage,
		stringToFind := "Previous generic diagnostic"
	),
	message := 'Omitting the borrowed entry message clears the previous prefix'
);
expect(
	condition := TOF_Core.WideStrings.Contains(
		stringToSearchIn := _AssertionRun.Assertion4.FailureMessage,
		stringToFind := "finite nonnegative comparison tolerance"
	),
	message := 'An invalid tolerance fails before a comparison that would otherwise pass'
);
expect(
	condition := _AssertionRun.Assertion14.Outcome = TOF_Testing.TEST_OUTCOME.PASSED,
	message := 'Independent context scenario CONTEXT_TRANSITIONS has its expected outcome'
);
expect(
	condition := _AssertionRun.Assertion15.Outcome = TOF_Testing.TEST_OUTCOME.FAILED,
	message := 'Independent context scenario TYPED_MESSAGE_AFTER_GENERIC has its expected outcome'
);
expect(
	condition := _AssertionRun.Assertion15.FailureMessage = "Independent typed: Expected: 11, but was: 10",
	message := 'Independent context scenario TYPED_MESSAGE_AFTER_GENERIC retains its diagnostic'
);
expect(
	condition := _AssertionRun.Assertion16.Outcome = TOF_Testing.TEST_OUTCOME.FAILED,
	message := 'Independent context scenario GENERIC_MESSAGE_AFTER_TYPED has its expected outcome'
);
expect(
	condition := _AssertionRun.Assertion16.FailureMessage = "Independent generic: Expected: 2, but was: 1",
	message := 'Independent context scenario GENERIC_MESSAGE_AFTER_TYPED retains its diagnostic'
);
expect(
	condition := _AssertionRun.Assertion17.Outcome = TOF_Testing.TEST_OUTCOME.FAILED,
	message := 'Independent context scenario TYPED_MESSAGE_RESET_AFTER_GENERIC has its expected outcome'
);
expect(
	condition := _AssertionRun.Assertion17.FailureMessage = "Expected: 2, but was: 1",
	message := 'Independent context scenario TYPED_MESSAGE_RESET_AFTER_GENERIC retains its diagnostic'
);
expect(
	condition := _AssertionRun.Assertion18.Outcome = TOF_Testing.TEST_OUTCOME.FAILED,
	message := 'Independent context scenario INTEGER_FAILURE has its expected outcome'
);
expect(
	condition := _AssertionRun.Assertion18.FailureMessage = "Expected: -2, but was: -3",
	message := 'Independent context scenario INTEGER_FAILURE retains its diagnostic'
);
expect(
	condition := _AssertionRun.Assertion19.Outcome = TOF_Testing.TEST_OUTCOME.FAILED,
	message := 'Independent context scenario BITSTRING_FAILURE has its expected outcome'
);
expect(
	condition := _AssertionRun.Assertion19.FailureMessage = "Expected: 11, but was: 10",
	message := 'Independent context scenario BITSTRING_FAILURE retains its diagnostic'
);
expect(
	condition := _AssertionRun.Assertion20.Outcome = TOF_Testing.TEST_OUTCOME.FAILED,
	message := 'Independent context scenario POINTER_FAILURE has its expected outcome'
);
expect(
	condition := TOF_Core.WideStrings.Contains(
		stringToSearchIn := _AssertionRun.Assertion20.FailureMessage,
		stringToFind := "Expected: 0, but was: "
	),
	message := 'Independent context scenario POINTER_FAILURE retains its diagnostic'
);
expect(
	condition := _AssertionRun.Assertion21.Outcome = TOF_Testing.TEST_OUTCOME.FAILED,
	message := 'Independent context scenario STRING_LONG_FAILURE has its expected outcome'
);
expect(
	condition := TOF_Core.WideStrings.Contains(
		stringToSearchIn := _AssertionRun.Assertion21.FailureMessage,
		stringToFind := "ASCII expected suffix"
	),
	message := 'Independent context scenario STRING_LONG_FAILURE retains its diagnostic'
);
expect(
	condition := _AssertionRun.Assertion22.Outcome = TOF_Testing.TEST_OUTCOME.FAILED,
	message := 'Independent context scenario WIDE_STRING_LONG_FAILURE has its expected outcome'
);
expect(
	condition := TOF_Core.WideStrings.Contains(
		stringToSearchIn := _AssertionRun.Assertion22.FailureMessage,
		stringToFind := "Wide expected suffix"
	),
	message := 'Independent context scenario WIDE_STRING_LONG_FAILURE retains its diagnostic'
);
expect(
	condition := _AssertionRun.Assertion23.Outcome = TOF_Testing.TEST_OUTCOME.FAILED,
	message := 'Independent context scenario STRING_CONTAINMENT_FAILURE has its expected outcome'
);
expect(
	condition := _AssertionRun.Assertion23.FailureMessage = "Expected text to contain 'missing', but was: 'present'",
	message := 'Independent context scenario STRING_CONTAINMENT_FAILURE retains its diagnostic'
);
expect(
	condition := _AssertionRun.Assertion24.Outcome = TOF_Testing.TEST_OUTCOME.FAILED,
	message := 'Independent context scenario FLOAT_ORDERING_FAILURE has its expected outcome'
);
expect(
	condition := TOF_Core.WideStrings.Contains(
		stringToSearchIn := _AssertionRun.Assertion24.FailureMessage,
		stringToFind := "Expected value > "
	),
	message := 'Independent context scenario FLOAT_ORDERING_FAILURE retains its diagnostic'
);
expect(
	condition := _AssertionRun.Assertion25.Outcome = TOF_Testing.TEST_OUTCOME.FAILED,
	message := 'Independent context scenario FLOAT_EQUALITY_FAILURE has its expected outcome'
);
expect(
	condition := TOF_Core.WideStrings.Contains(
		stringToSearchIn := _AssertionRun.Assertion25.FailureMessage,
		stringToFind := ", tolerance: "
	),
	message := 'Independent context scenario FLOAT_EQUALITY_FAILURE retains its diagnostic'
);
expect(
	condition := _AssertionRun.Assertion26.Outcome = TOF_Testing.TEST_OUTCOME.FAILED,
	message := 'Independent context scenario TIME_ORDERING_FAILURE has its expected outcome'
);
expect(
	condition := TOF_Core.WideStrings.Contains(
		stringToSearchIn := _AssertionRun.Assertion26.FailureMessage,
		stringToFind := "Expected value >= "
	),
	message := 'Independent context scenario TIME_ORDERING_FAILURE retains its diagnostic'
);
checkAssertionContracts := TRUE;
END_METHOD

(*!
<summary>Checks assertion and direct failure routing between independent active cases.</summary>
<description>Configures the persistent output probes through local references without copying them.
Returns TRUE when all observations for this scenario are complete.
</description>
*)
METHOD PRIVATE checkCaseIsolation : BOOL
VAR
	passingProbe : REFERENCE TO AssertionIsolationProbe;
	failingProbe : REFERENCE TO AssertionIsolationProbe;
END_VAR
passingProbe REF= _PassingRun.Child;
failingProbe REF= _FailingRun.Child;

IF NOT _IsolationConfigured THEN
	passingProbe.Peer := ADR(failingProbe);
	failingProbe.Timeout := T#0S;
	passingProbe.Timeout := T#0S;
	_FailingRun.Reporter := _FailureReport;
	_PassingRun.Reporter := _PassReport;
	_IsolationConfigured := TRUE;
END_IF

_FailingRun.Execute(cleanupTaskMemory := FALSE);
_PassingRun.Execute(cleanupTaskMemory := FALSE);
_IsolationCalls := _IsolationCalls + 1;

IF NOT (_FailingRun.IsFinished AND_THEN _PassingRun.IsFinished) AND_THEN _IsolationCalls < 16 THEN
	RETURN;
END_IF

expect(condition := _FailingRun.IsFinished AND _PassingRun.IsFinished, message := 'Both runs finish');
expectDInt(expected := 1, actual := _FailingRun.FailedTests, message := 'Failure belongs to receiver');
expectDInt(expected := 1, actual := _PassingRun.PassedTests, message := 'Calling case passes');
expectDInt(expected := 0, actual := _PassingRun.FailedTests, message := 'Calling case has no peer failure');

IF NOT _IsolationSecondRun AND_THEN _FailingRun.IsFinished AND_THEN _PassingRun.IsFinished THEN
	_IsolationSecondRun := TRUE;
	passingProbe.UseDirectFailure := TRUE;
	_IsolationCalls := 0;
	_FailingRun.Reset();
	_PassingRun.Reset();
	RETURN;
END_IF

checkCaseIsolation := TRUE;
END_METHOD

(*!
<summary>Checks all typed contexts through IObject before assertion preparation.</summary>
<description>
Persistent contexts retain their default state. Checks metadata, addresses and inherited identity equality;
no test callback or Prepare call is required to read Object metadata.
Also checks concrete runner metadata, the inherited INamed signature and the constructor-copied group name.
Context namespaces are compared with an independent library reporter; runner metadata uses the consumer namespace.

Returns TRUE when all observations for this scenario are complete.
</description>
*)
METHOD PRIVATE checkContextObjects : BOOL
VAR
	first : TOF_Core.IObject;
	second : TOF_Core.IObject;
	group : TOF_Core.IObject;
	named : TOF_Core.INamed;
	displayName : REFERENCE TO WSTRING;
	concreteDisplayName : REFERENCE TO WSTRING;
END_VAR
assertObjectMetadata(
	object := _Runner,
	expectedNamespaceName := CurrentNamespace.Name,
	expectedClassName := 'MixedTestRunner',
	expectedSize := XSIZEOF(_Runner),
	expectedAddress := ADR(_Runner)
);

assertObjectMetadata(
	object := _MetadataBoolAssertionContext,
	expectedNamespaceName := _ExceptionAdsReporter.NamespaceName,
	expectedClassName := 'BoolAssertionContext',
	expectedSize := XSIZEOF(_MetadataBoolAssertionContext),
	expectedAddress := ADR(_MetadataBoolAssertionContext)
);
assertObjectMetadata(
	object := _MetadataByteAssertionContext,
	expectedNamespaceName := _ExceptionAdsReporter.NamespaceName,
	expectedClassName := 'ByteAssertionContext',
	expectedSize := XSIZEOF(_MetadataByteAssertionContext),
	expectedAddress := ADR(_MetadataByteAssertionContext)
);
assertObjectMetadata(
	object := _MetadataDateAssertionContext,
	expectedNamespaceName := _ExceptionAdsReporter.NamespaceName,
	expectedClassName := 'DateAssertionContext',
	expectedSize := XSIZEOF(_MetadataDateAssertionContext),
	expectedAddress := ADR(_MetadataDateAssertionContext)
);
assertObjectMetadata(
	object := _MetadataDateTimeAssertionContext,
	expectedNamespaceName := _ExceptionAdsReporter.NamespaceName,
	expectedClassName := 'DateTimeAssertionContext',
	expectedSize := XSIZEOF(_MetadataDateTimeAssertionContext),
	expectedAddress := ADR(_MetadataDateTimeAssertionContext)
);
assertObjectMetadata(
	object := _MetadataDIntAssertionContext,
	expectedNamespaceName := _ExceptionAdsReporter.NamespaceName,
	expectedClassName := 'DIntAssertionContext',
	expectedSize := XSIZEOF(_MetadataDIntAssertionContext),
	expectedAddress := ADR(_MetadataDIntAssertionContext)
);
assertObjectMetadata(
	object := _MetadataDWordAssertionContext,
	expectedNamespaceName := _ExceptionAdsReporter.NamespaceName,
	expectedClassName := 'DWordAssertionContext',
	expectedSize := XSIZEOF(_MetadataDWordAssertionContext),
	expectedAddress := ADR(_MetadataDWordAssertionContext)
);
assertObjectMetadata(
	object := _MetadataIntAssertionContext,
	expectedNamespaceName := _ExceptionAdsReporter.NamespaceName,
	expectedClassName := 'IntAssertionContext',
	expectedSize := XSIZEOF(_MetadataIntAssertionContext),
	expectedAddress := ADR(_MetadataIntAssertionContext)
);
assertObjectMetadata(
	object := _MetadataLIntAssertionContext,
	expectedNamespaceName := _ExceptionAdsReporter.NamespaceName,
	expectedClassName := 'LIntAssertionContext',
	expectedSize := XSIZEOF(_MetadataLIntAssertionContext),
	expectedAddress := ADR(_MetadataLIntAssertionContext)
);
assertObjectMetadata(
	object := _MetadataLongDateAssertionContext,
	expectedNamespaceName := _ExceptionAdsReporter.NamespaceName,
	expectedClassName := 'LongDateAssertionContext',
	expectedSize := XSIZEOF(_MetadataLongDateAssertionContext),
	expectedAddress := ADR(_MetadataLongDateAssertionContext)
);
assertObjectMetadata(
	object := _MetadataLongDateTimeAssertionContext,
	expectedNamespaceName := _ExceptionAdsReporter.NamespaceName,
	expectedClassName := 'LongDateTimeAssertionContext',
	expectedSize := XSIZEOF(_MetadataLongDateTimeAssertionContext),
	expectedAddress := ADR(_MetadataLongDateTimeAssertionContext)
);
assertObjectMetadata(
	object := _MetadataLongRealAssertionContext,
	expectedNamespaceName := _ExceptionAdsReporter.NamespaceName,
	expectedClassName := 'LongRealAssertionContext',
	expectedSize := XSIZEOF(_MetadataLongRealAssertionContext),
	expectedAddress := ADR(_MetadataLongRealAssertionContext)
);
assertObjectMetadata(
	object := _MetadataLongTimeAssertionContext,
	expectedNamespaceName := _ExceptionAdsReporter.NamespaceName,
	expectedClassName := 'LongTimeAssertionContext',
	expectedSize := XSIZEOF(_MetadataLongTimeAssertionContext),
	expectedAddress := ADR(_MetadataLongTimeAssertionContext)
);
assertObjectMetadata(
	object := _MetadataLongTimeOfDayAssertionContext,
	expectedNamespaceName := _ExceptionAdsReporter.NamespaceName,
	expectedClassName := 'LongTimeOfDayAssertionContext',
	expectedSize := XSIZEOF(_MetadataLongTimeOfDayAssertionContext),
	expectedAddress := ADR(_MetadataLongTimeOfDayAssertionContext)
);
assertObjectMetadata(
	object := _MetadataLWordAssertionContext,
	expectedNamespaceName := _ExceptionAdsReporter.NamespaceName,
	expectedClassName := 'LWordAssertionContext',
	expectedSize := XSIZEOF(_MetadataLWordAssertionContext),
	expectedAddress := ADR(_MetadataLWordAssertionContext)
);
assertObjectMetadata(
	object := _MetadataPointerAssertionContext,
	expectedNamespaceName := _ExceptionAdsReporter.NamespaceName,
	expectedClassName := 'PointerAssertionContext',
	expectedSize := XSIZEOF(_MetadataPointerAssertionContext),
	expectedAddress := ADR(_MetadataPointerAssertionContext)
);
assertObjectMetadata(
	object := _MetadataRealAssertionContext,
	expectedNamespaceName := _ExceptionAdsReporter.NamespaceName,
	expectedClassName := 'RealAssertionContext',
	expectedSize := XSIZEOF(_MetadataRealAssertionContext),
	expectedAddress := ADR(_MetadataRealAssertionContext)
);
assertObjectMetadata(
	object := _MetadataSIntAssertionContext,
	expectedNamespaceName := _ExceptionAdsReporter.NamespaceName,
	expectedClassName := 'SIntAssertionContext',
	expectedSize := XSIZEOF(_MetadataSIntAssertionContext),
	expectedAddress := ADR(_MetadataSIntAssertionContext)
);
assertObjectMetadata(
	object := _MetadataStringAssertionContext,
	expectedNamespaceName := _ExceptionAdsReporter.NamespaceName,
	expectedClassName := 'StringAssertionContext',
	expectedSize := XSIZEOF(_MetadataStringAssertionContext),
	expectedAddress := ADR(_MetadataStringAssertionContext)
);
assertObjectMetadata(
	object := _MetadataTimeAssertionContext,
	expectedNamespaceName := _ExceptionAdsReporter.NamespaceName,
	expectedClassName := 'TimeAssertionContext',
	expectedSize := XSIZEOF(_MetadataTimeAssertionContext),
	expectedAddress := ADR(_MetadataTimeAssertionContext)
);
assertObjectMetadata(
	object := _MetadataTimeOfDayAssertionContext,
	expectedNamespaceName := _ExceptionAdsReporter.NamespaceName,
	expectedClassName := 'TimeOfDayAssertionContext',
	expectedSize := XSIZEOF(_MetadataTimeOfDayAssertionContext),
	expectedAddress := ADR(_MetadataTimeOfDayAssertionContext)
);
assertObjectMetadata(
	object := _MetadataUDIntAssertionContext,
	expectedNamespaceName := _ExceptionAdsReporter.NamespaceName,
	expectedClassName := 'UDIntAssertionContext',
	expectedSize := XSIZEOF(_MetadataUDIntAssertionContext),
	expectedAddress := ADR(_MetadataUDIntAssertionContext)
);
assertObjectMetadata(
	object := _MetadataUIntAssertionContext,
	expectedNamespaceName := _ExceptionAdsReporter.NamespaceName,
	expectedClassName := 'UIntAssertionContext',
	expectedSize := XSIZEOF(_MetadataUIntAssertionContext),
	expectedAddress := ADR(_MetadataUIntAssertionContext)
);
assertObjectMetadata(
	object := _MetadataULIntAssertionContext,
	expectedNamespaceName := _ExceptionAdsReporter.NamespaceName,
	expectedClassName := 'ULIntAssertionContext',
	expectedSize := XSIZEOF(_MetadataULIntAssertionContext),
	expectedAddress := ADR(_MetadataULIntAssertionContext)
);
assertObjectMetadata(
	object := _MetadataUSIntAssertionContext,
	expectedNamespaceName := _ExceptionAdsReporter.NamespaceName,
	expectedClassName := 'USIntAssertionContext',
	expectedSize := XSIZEOF(_MetadataUSIntAssertionContext),
	expectedAddress := ADR(_MetadataUSIntAssertionContext)
);
assertObjectMetadata(
	object := _MetadataWideStringAssertionContext,
	expectedNamespaceName := _ExceptionAdsReporter.NamespaceName,
	expectedClassName := 'WideStringAssertionContext',
	expectedSize := XSIZEOF(_MetadataWideStringAssertionContext),
	expectedAddress := ADR(_MetadataWideStringAssertionContext)
);
assertObjectMetadata(
	object := _MetadataWordAssertionContext,
	expectedNamespaceName := _ExceptionAdsReporter.NamespaceName,
	expectedClassName := 'WordAssertionContext',
	expectedSize := XSIZEOF(_MetadataWordAssertionContext),
	expectedAddress := ADR(_MetadataWordAssertionContext)
);

first := _MetadataBoolAssertionContext;
second := _OtherBoolContext;
expect(condition := first.Equals(other := first), message := 'A context equals itself');
expectFalse(condition := first.Equals(other := second), message := 'Equal snapshots do not merge context identity');
expectFalse(condition := first.Equals(other := 0), message := 'A context is distinct from null');

group := _Runner.Empty;
expect(condition := group.ClassName <> '', message := 'A concrete group provides its class name');
expect(
	condition := group.NamespaceName = _Runner.NamespaceName,
	message := 'Group and runner share the consumer namespace'
);
expect(condition := group.SelfSize = XSIZEOF(_Runner.Empty), message := 'Group size includes its concrete storage');
expect(
	condition := group.SelfAddress = ADR(_Runner.Empty),
	message := 'Group identity points to the concrete instance'
);

named := _Runner.Empty;
displayName REF= named.Name;
concreteDisplayName REF= _Runner.Empty.Name;
expect(condition := __ISVALIDREF(displayName), message := 'INamed provides a valid name reference');
expect(condition := ADR(displayName) = ADR(concreteDisplayName), message := 'INamed borrows the same name storage');
expect(condition := displayName = "Empty", message := 'INamed exposes the constructor-copied group name');

checkContextObjects := TRUE;
END_METHOD

(*!
<summary>Checks deadline completion, BUSY failure termination and mutation guards.</summary>
<description>
Configures the persistent output leaf through a local reference without copying it.
The first run must exercise active mutation guards before the deadline. The second injects a BUSY failure.
Returns TRUE when all observations for this scenario are complete.
</description>
*)
METHOD PRIVATE checkDeadline : BOOL
VAR
	deadlineProbe : REFERENCE TO AssertionIsolationProbe;
	exceptionCode : __SYSTEM.ExceptionCode;
	rejected : BOOL;
	actualParent : TOF_Testing.ITestElement;
END_VAR
deadlineProbe REF= _DeadlineRun.DeadlineGroup.Child;

IF NOT _DeadlineConfigured THEN
	deadlineProbe.CompleteAfterCycle := 0;
	deadlineProbe.Timeout := T#1MS;
	_DeadlineRun.Reporter := _DeadlineReport;
	_DeadlineConfigured := TRUE;
END_IF

_DeadlineRun.Execute(cleanupTaskMemory := FALSE);
_DeadlineCalls := _DeadlineCalls + 1;

IF deadlineProbe.IsRunning AND_THEN NOT _DeadlineBusyFailureRun AND_THEN NOT _ActiveConfigurationChecked THEN

	__TRY
		deadlineProbe.Timeout := T#2S;
	__CATCH(exceptionCode)
		assertCaughtExceptionType(
			exceptionCode := exceptionCode,
			expectedTypeName := 'StandardException'
		);
		rejected := TRUE;
	__ENDTRY

	expect(condition := rejected, message := 'An active deadline cannot be changed');
	expect(
		condition := deadlineProbe.Timeout = T#1MS,
		message := 'Rejected mutation preserves the deadline'
	);
	_DeadlineRun.Reset();
	expect(
		condition := deadlineProbe.IsRunning AND_THEN NOT _DeadlineRun.IsFinished,
		message := 'Active Reset leaves the pending leaf running'
	);
	rejected := FALSE;

	__TRY
		_DeadlineRun.Reporter := _DeadlineReport;
	__CATCH(exceptionCode)
		assertCaughtExceptionType(
			exceptionCode := exceptionCode,
			expectedTypeName := 'StandardException'
		);
		rejected := TRUE;
	__ENDTRY

	expect(condition := rejected, message := 'Active runner rejects Reporter mutation');
	actualParent := deadlineProbe.Parent;
	expect(
		condition := actualParent = _DeadlineRun.Children[0],
		message := 'The active leaf retains its constructor-assigned parent'
	);
	_ActiveConfigurationChecked := TRUE;
END_IF

IF NOT _DeadlineRun.IsFinished AND_THEN _DeadlineCalls < _DeadlineScanLimit THEN
	RETURN;
END_IF

IF NOT _DeadlineBusyFailureRun THEN
	expect(condition := _DeadlineRun.IsFinished, message := 'A one-millisecond nominal deadline terminates');
	expect(condition := _ActiveConfigurationChecked, message := 'Deadline run exercises the active mutation guards');
	expectDInt(expected := 1, actual := _DeadlineRun.FailedTests, message := 'Deadline is one failed leaf');
	expectUDInt(
		expected := 1,
		actual := deadlineProbe.TeardownCalls,
		message := 'Deadline cleanup occurs once'
	);

	IF _DeadlineRun.IsFinished THEN
		_DeadlineBusyFailureRun := TRUE;
		_DeadlineCalls := 0;
		_DeadlineRun.Reset();
		deadlineProbe.Timeout := T#0S;
		deadlineProbe.FailSelfWhileBusy := TRUE;
		RETURN;
	END_IF
ELSE
	expect(condition := _DeadlineRun.IsFinished, message := 'A failed BUSY step terminates immediately');
	expectDInt(expected := 1, actual := _DeadlineRun.FailedTests, message := 'BUSY failure counts once');
	expectUDInt(
		expected := 1,
		actual := deadlineProbe.BodyCalls,
		message := 'Failed BUSY step does not run another body cycle'
	);
	expectUDInt(
		expected := 1,
		actual := deadlineProbe.TeardownCalls,
		message := 'Failed BUSY cleanup occurs once'
	);
END_IF

checkDeadline := TRUE;
END_METHOD

(*!
<summary>Checks copied native, fallback and long diagnostics after earlier task-cycle cleanup.</summary>
<description>
Requires the inner run to finish and publish its report before the suite accepts the diagnostic results.
Returns TRUE when all observations for this scenario are complete.
</description>
*)
METHOD PRIVATE checkDiagnostics : BOOL
VAR
	probe : REFERENCE TO DiagnosticProbe;
END_VAR
IF NOT _DiagnosticConfigured THEN
	probe REF= _DiagnosticRun.NativeDiagnostic;
	probe.ThrowNative := TRUE;
	probe REF= _DiagnosticRun.FormatterDiagnostic;
	probe.ThrowOnGetMessage := TRUE;
	_DiagnosticRun.Reporter := _DiagnosticReport;
	_DiagnosticConfigured := TRUE;
END_IF

_DiagnosticRun.Execute(cleanupTaskMemory := FALSE);
_DiagnosticCalls := _DiagnosticCalls + 1;

IF NOT _DiagnosticRun.IsFinished AND_THEN _DiagnosticCalls < 16 THEN
	RETURN;
END_IF

expect(condition := _DiagnosticRun.IsFinished, message := 'The diagnostic run finishes within 16 scans');
expect(condition := _DiagnosticReport.IsReady, message := 'The diagnostic report is complete');
expectDInt(
	expected := 3,
	actual := _DiagnosticRun.FailedTests,
	message := 'All injected errors are failed leaves'
);
expect(
	condition := TOF_Core.WideStrings.Contains(stringToSearchIn := _DiagnosticRun.NativeDiagnostic.FailureMessage,
		stringToFind := "ExecuteTest"),
	message := 'Native diagnostic has the interrupted stage'
);
expect(
	condition := TOF_Core.WideStrings.Contains(stringToSearchIn := _DiagnosticRun.FormatterDiagnostic.FailureMessage,
		stringToFind := "diagnostic unavailable"),
	message := 'Failing GetMessage retains stage/code fallback'
);
expect(
	condition := TOF_Core.WideStrings.Contains(stringToSearchIn := _DiagnosticRun.LongDiagnostic.FailureMessage,
		stringToFind := "END_OF_LONG_DIAGNOSTIC"),
	message := 'Long copied exception message is not narrowed to 255'
);
expectUDInt(
	expected := 1,
	actual := _DiagnosticRun.FormatterDiagnostic.TeardownCalls,
	message := 'Fallback still tears down once'
);
checkDiagnostics := TRUE;
END_METHOD

(*!
<summary>Checks a zero-child runner completes successfully with zero tests.</summary>
<description>Returns TRUE when all observations for this scenario are complete.</description>
*)
METHOD PRIVATE checkEmptyRun : BOOL
IF NOT _EmptyConfigured THEN
	_EmptyRun.Reporter := _EmptyReport;
	_EmptyConfigured := TRUE;
END_IF

_EmptyRun.Execute(cleanupTaskMemory := FALSE);
_EmptyCalls := _EmptyCalls + 1;

IF NOT _EmptyRun.IsFinished AND_THEN _EmptyCalls < _EmptyScanLimit THEN
	RETURN;
END_IF

expect(condition := _EmptyRun.IsFinished, message := 'An empty run must finish within the scan limit');
expect(condition := _EmptyRun.AllPassed, message := 'An empty run passes');
expectDInt(expected := 0, actual := _EmptyRun.TotalTests, message := 'No synthetic empty test');
checkEmptyRun := TRUE;
END_METHOD

(*!
<summary>Checks missing static storage, safe abort recovery rejection and invalid reporter outcomes.</summary>
<description>Returns TRUE when all observations for this scenario are complete.</description>
*)
METHOD PRIVATE checkExceptionClasses : BOOL
VAR
	exceptionCode : __SYSTEM.ExceptionCode;
	rejected : BOOL;
	diagnostic : TOF_Core.ERROR_MESSAGE;
END_VAR
__TRY
	_MissingConfigurationGroup.Reset(reporter := 0);
__CATCH(exceptionCode)
	assertCaughtExceptionType(exceptionCode := exceptionCode, expectedTypeName := 'DataMemberNotSpecifiedException');
	rejected := TRUE;
__ENDTRY

expect(condition := rejected, message := 'Group Reset rejects missing child-array storage');
_MissingConfigurationRunner.Execute(cleanupTaskMemory := FALSE);
expectDInt(
	expected := -1,
	actual := _MissingConfigurationRunner.ExitCode,
	message := 'Missing runner storage aborts'
);
assertCaughtExceptionType(
	exceptionCode := _MissingConfigurationRunner.CallbackException,
	expectedTypeName := 'DataMemberNotSpecifiedException'
);
rejected := FALSE;

__TRY
	_MissingConfigurationRunner.Reset();
__CATCH(exceptionCode)
	assertCaughtExceptionType(exceptionCode := exceptionCode, expectedTypeName := 'DataMemberNotSpecifiedException');
	rejected := TRUE;
__ENDTRY

